IF (seq.Step(inStepID := seq.RESTORE_STEP_ID,
    inEnabled := TRUE,
    inStepDescription := 'RETURN TO THE START OF THE SEQUENCE')) THEN
    //--------------------------------------------------------	
		refSequenceTask.DoneWhen(TRUE);
    	seq.CompleteSequence();
    //--------------------------------------------------------			
END_IF;


IF refSequenceTask.HandleTaskError() THEN
	//here we can decide what to do
	//	refSequenceTask.Restore();
	_feedNewBlisterTask.Restore();
END_IF



seq.Close();
END_METHOD

METHOD PRIVATE SequenceOutgoingBlister
VAR_INPUT
	refSequenceTask : REFERENCE TO TcoFeedingSequenceTask;
	
	
END_VAR

VAR
    seq    : REFERENCE TO TcoCore.TcoSequence;

END_VAR

VAR_INST
	_timer:ton;
	
END_VAR
seq REF= refSequenceTask.Sequence;
refSequenceTask(inoStatus:=_status,inoConfig:=_config);

seq.Open();
seq.Observer := refSequenceTask.Observer;



		



//***************************************************************************************************     
//    This step will be executed and immediately finished, as the condition in Await method is true.
IF seq.Step(0,TRUE,'<#INIT#>') THEN   
	Messenger.Warning('<#BEZPECNOST ZARIADENIA NARUSENA. NIEJE MOZNE VYKONAT AKCIU#>');     
	IF _status.SafeCondition THEN
    	seq.CompleteStep();
	END_IF;
END_IF        
//***************************************************************************************************     

IF seq.Step(10,TRUE,'<#SEPAROVANIE VYSTUPNEHO BLISTRA - UVOLNENIE BLISTRA VYSUNUTIE P9#>') THEN   

    seq.StepCompleteWhen( (THIS^.Components.P9_LockEntryBlisterTop.MoveToWork().Done OR _config.LockBlisterInPickPosInactive) AND THIS^.Components.P8_FixEntryBlisterSide.MoveToHome().Done);
END_IF        
//***************************************************************************************************   


//***************************************************************************************************     
IF seq.Step(20,TRUE,'<#SEPAROVANIE VYSTUPNEHO BLISTRA - ZASUNUTIE SUPPORTU P7#>') THEN   

   seq.StepCompleteWhen(THIS^.Components.P7_SupportEntryBlister.MoveToHome().Done);
END_IF        
//***************************************************************************************************   



//***************************************************************************************************     
IF seq.Step(30,TRUE,'<#SEPAROVANIE VYSTUPNEHO BLISTRA - KONTROLA PRITOMNOSTI BLISTA NA SKLZE (I5) #>') THEN   
	IF seq.IsFreshState THEN
		_timer(IN:=FALSE);
	END_IF
	_timer(IN:=THIS^.Components.I5_OutBlistersIsThrowedCorrectly.Signal,PT:=_config.StabilisationTime);
	
    seq.StepCompleteWhen(_timer.Q);
	
	IF Components.P4_FeedEntryBlister.AtHome AND NOT THIS^.Components.I5_OutBlistersIsThrowedCorrectly.Signal THEN
		seq.StepCompleteWhen(seq.CurrentStep.Duration>_config.StabilisationTime);
	END_IF
END_IF        
//***************************************************************************************************   



IF (seq.Step(inStepID := seq.RESTORE_STEP_ID,
    inEnabled := TRUE,
    inStepDescription := 'RETURN TO THE START OF THE SEQUENCE')) THEN
    //--------------------------------------------------------	
		refSequenceTask.DoneWhen(TRUE);
    	seq.CompleteSequence();
    //--------------------------------------------------------			
END_IF;


IF refSequenceTask.HandleTaskError() THEN
	//here we can decide what to do
	//	refSequenceTask.Restore();
	_throwBlisterTask.Restore();


END_IF


seq.Close();
END_METHOD

METHOD PRIVATE SequenceOutgoingBuffer
VAR_INPUT
	refSequenceTask : REFERENCE TO TcoFeedingSequenceTask;
	
	
END_VAR

VAR
    seq    : REFERENCE TO TcoCore.TcoSequence;

END_VAR

VAR_INST
	_timer:ton;
	
END_VAR
seq REF= refSequenceTask.Sequence;
refSequenceTask(inoStatus:=_status,inoConfig:=_config);

seq.Open();
seq.Observer := refSequenceTask.Observer;



		



//***************************************************************************************************     
//    This step will be executed and immediately finished, as the condition in Await method is true.
IF seq.Step(0,TRUE,'<#INIT#>') THEN   
	Messenger.Warning('<#BEZPECNOST ZARIADENIA NARUSENA. NIEJE MOZNE VYKONAT AKCIU#>');     
	IF _status.SafeCondition THEN
    	seq.CompleteStep();
	END_IF;
END_IF        
//***************************************************************************************************     



//***************************************************************************************************     
IF seq.Step(10,TRUE,'<#VYSTUPNY BUFFER - KONTROLA PRITOMNOSTI BLISTA NAD BUFFEROM  #>') THEN   
	IF seq.IsFreshState THEN
		_timer(IN:=FALSE);
	END_IF
	_timer(IN:=(*NOT THIS^.Components.I5_OutBlistersIsThrowedCorrectly.Signal AND*) Components.I7_OutBlistersIsAboveOutBuffer.Signal,PT:=_config.StabilisationTime);
	
    seq.StepCompleteWhen(_timer.Q);
END_IF        
//***************************************************************************************************   


//***************************************************************************************************     
IF seq.Step(20,TRUE,'<#VYSTUPNY BUFFER - KONTROLA POSCTU BLISTROV SNIMAC I8 #>') THEN   
	Messenger.Warning('<#PODAVAC PLNY! ODSTRANTE PRAZDNE BLISTRE (I8) !#>');
    seq.StepCompleteWhen(THIS^.Components.I8_OutBlistersBufferIsFull.IsFalse);
END_IF        
//***************************************************************************************************   


//***************************************************************************************************     
IF seq.Step(30,TRUE,'<#VYSTUPNY BUFFER - P6 POSUN KUSOV NAD BUFFER#>') THEN   

	THIS^.Components.P6_VerticalSepareOutBlister.MoveToWork();
	IF Components.I6_OutBlistersLisftSignal.Signal THEN
	
		THIS^.Components.P6_VerticalSepareOutBlister.MoveWorkTask.Abort();
	    seq.StepCompleteWhen(TRUE);
	END_IF;
		
END_IF        
//***************************************************************************************************   


//***************************************************************************************************     
IF seq.Step(40,TRUE,'<#VYSTUPNY BUFFER - UVOLNENIE BLISTRA  P5 PRACOVNA POZICIA #>') THEN   

	
	seq.StepCompleteWhen(Components.P5_HorizontalSepareOutBlisters.MoveToWork().Done);
		
END_IF        
//***************************************************************************************************   

//***************************************************************************************************     
IF seq.Step(45,TRUE,'<#VYSTUPNY BUFFER - P6 NAVRAT NAHOR#>') THEN   

	
	seq.StepCompleteWhen( THIS^.Components.P6_VerticalSepareOutBlister.MoveToHome().Done);
		
END_IF        
//***************************************************************************************************   

//***************************************************************************************************     
IF seq.Step(50,TRUE,'<#VYSTUPNY BUFFER - HORIZONTALNE ZASUNUTIE P5 ZAKLADNA POZICIA#>') THEN   

	
	seq.StepCompleteWhen(Components.P5_HorizontalSepareOutBlisters.MoveToHome().Done);
		
END_IF        
//***************************************************************************************************   



IF (seq.Step(inStepID := seq.RESTORE_STEP_ID,
    inEnabled := TRUE,
    inStepDescription := 'RETURN TO THE START OF THE SEQUENCE')) THEN
    //--------------------------------------------------------	
		refSequenceTask.DoneWhen(TRUE);
    	seq.CompleteSequence();
    //--------------------------------------------------------			
END_IF;


IF refSequenceTask.HandleTaskError() THEN
	//here we can decide what to do
	//refSequenceTask.Restore();
	_hanldeOutBufferTask.Restore();
END_IF


seq.Close();
END_METHOD

METHOD PRIVATE SequenceResetToDefault
VAR_INPUT
	refSequenceTask : REFERENCE TO TcoFeedingSequenceTask;
	
	
END_VAR

VAR
    seq    : REFERENCE TO TcoCore.TcoSequence;

END_VAR

VAR_INST
	_timer:ton;
	
END_VAR
seq REF= refSequenceTask.Sequence;
refSequenceTask(inoStatus:=_status,inoConfig:=_config);
seq.Open();
seq.Observer := refSequenceTask.Observer;



		



//***************************************************************************************************     
//    This step will be executed and immediately finished, as the condition in Await method is true.
IF seq.Step(0,TRUE,'<#INIT#>') THEN   
	Messenger.Warning('<#BEZPECNOST ZARIADENIA NARUSENA. NIEJE MOZNE VYKONAT AKCIU#>');     
	IF _status.SafeCondition THEN
    	seq.CompleteStep();
	END_IF;
END_IF        
//***************************************************************************************************     



//***************************************************************************************************     
IF seq.Step(10,TRUE,'<#VYCHODIZA POLOHA - VYSUNUTIE P3#>') THEN   

    seq.StepCompleteWhen(Components.P3_HorizontalSepareEntryBlisters.MoveToWork().Done );
END_IF        
//***************************************************************************************************   


//***************************************************************************************************     
IF seq.Step(20,NOT _config.SepareBlistersAtEntryInactive,'<#VYCHODIZA POLOHA - ZASUNUTIE P10#>') THEN   

    seq.StepCompleteWhen(Components.P10_HoldEntrySepareOutBlister.MoveToHome().Done);
END_IF        
//***************************************************************************************************   


//***************************************************************************************************     
IF seq.Step(30,TRUE,'<#VYCHODIZA POLOHA - ZASUNUTIE P1 A P2>') THEN   


	    seq.StepCompleteWhen(Components.P1_VerticalSepareEntryBlisters.MoveToHome().Done AND_THEN Components.P2_VerticalSepareEntryBlisters.MoveToHome().Done);

END_IF        
//***************************************************************************************************   


//***************************************************************************************************     
IF seq.Step(40,TRUE,'<#VYCHODIZA POLOHA - ZASUNUTIE P5#>') THEN   

	
	seq.StepCompleteWhen(Components.P5_HorizontalSepareOutBlisters.MoveToHome().Done);
		
END_IF        
//***************************************************************************************************   

//***************************************************************************************************     
IF seq.Step(50,TRUE,'<#VYCHODIZA POLOHA - ZASUNUTIE P6#>') THEN   

	
	seq.StepCompleteWhen(Components.P6_VerticalSepareOutBlister.MoveToHome().Done);
		
END_IF        
//***************************************************************************************************   

//***************************************************************************************************     
IF seq.Step(60,TRUE,'<#VYCHODIZA POLOHA - ZASUNUTIE P4 DO ZAKLADNEJ POZICIE#>') THEN   

	
	seq.StepCompleteWhen(Components.P4_FeedEntryBlister.MoveToHome().Done);
		
END_IF        
//***************************************************************************************************   

//***************************************************************************************************     
IF seq.Step(70,COmponents.I4_PresentBlisterInWorkingPos.Signal AND
				Components.P8_FixEntryBlisterSide.AtWork,'<#SEPAROVANIE VSTUPNEHO BLISTRA - PODoPRETIE  A ZAFIXOVANIE KUSU P7 VYSUNT A P9 ZASUNUT #>') THEN   

    seq.StepCompleteWhen(THIS^.Components.P7_SupportEntryBlister.MoveToWork().Done AND (THIS^.Components.P9_LockEntryBlisterTop.MoveToHome().Done OR _config.LockBlisterInPickPosInactive));
END_IF        
//***************************************************************************************************   


IF (seq.Step(inStepID := seq.RESTORE_STEP_ID,
    inEnabled := TRUE,
    inStepDescription := 'RETURN TO THE START OF THE SEQUENCE')) THEN
    //--------------------------------------------------------	
		refSequenceTask.DoneWhen(TRUE);
    	seq.CompleteSequence();
    //--------------------------------------------------------			
END_IF;



IF refSequenceTask.HandleTaskError() THEN
	
	//here we can decide what to do
	//	refSequenceTask.Restore();

END_IF

seq.Close();
END_METHOD

(*~
	<docu>
		<summary>
		    Custom service (manual, maintenance) logic.
			This method must be implemented in derived class.
		</summary>			
	</docu>	
~*)
METHOD PROTECTED  ServiceMode
_components.Q3_AttentionSignalisationB.Service();
_components.Q2_AttentionSignalisationG.Service();
_components.Q1_AttentionSignalisationR.Service();
_components.P1_VerticalSepareEntryBlisters.Service();
_components.P2_VerticalSepareEntryBlisters.Service();
_components.P3_HorizontalSepareEntryBlisters.Service();
_components.P4_FeedEntryBlister.Service();
_components.P5_HorizontalSepareOutBlisters.Service();
_components.P6_VerticalSepareOutBlister.Service();
_components.P7_SupportEntryBlister.Service();
_components.P8_FixEntryBlisterSide.Service();
_components.P9_LockEntryBlisterTop.Service();
_components.P10_HoldEntrySepareOutBlister.Service();
END_METHOD

PROPERTY PUBLIC SetSequencesToStep : bool
GET
SetSequencesToStep:=_setSequencesToStep;
END_GET
SET
_setSequencesToStep:=SetSequencesToStep;
END_SET
END_PROPERTY

METHOD PUBLIC SetToDefault : TcoCore.ITcoTaskStatus
SetToDefault := _setToDefaultTask.Invoke();
END_METHOD

PROPERTY SetToDefaultTask : REFERENCE TO TcoFeedingSequenceTask
GET
SetToDefaultTask ref=_setToDefaultTask;
END_GET
END_PROPERTY

(*~
	<docu>
		<summary>
			Gets the status of the MTS Pls feeder. 					
		</summary>			
	</docu>	
~*)
PROPERTY Status : REFERENCE TO TcoPlsPaletizator_Status_v_1_x_x
GET
Status REF= _status;
END_GET
END_PROPERTY

METHOD PUBLIC ThrowBlister : TcoCore.ITcoTaskStatus

ThrowBlister := _throwBlisterTask.Invoke();
END_METHOD

PROPERTY ThrowBlisterTask : REFERENCE TO TcoFeedingSequenceTask
GET
ThrowBlisterTask ref=_throwBlisterTask;
END_GET
END_PROPERTY

END_FUNCTION_BLOCK

// ---- Abstractions/Components/MtsFeeding/Components/OscilatingConveyorFeeder/TcoOscilatingConveyorFeeder.TcPOU
FUNCTION_BLOCK TcoOscilatingConveyorFeeder EXTENDS TcoCore.TcoComponent
VAR_INPUT
    inSafeCondition : BOOL;
    inDoorOpen : BOOL;
    inMOde : eCUMode;
END_VAR

VAR_OUTPUT
END_VAR
VAR
    {attribute addProperty Name "<#Config#>"}
    _config : TcoOscilatingConveyorFeeder_Config_v_1_x_x;
    {attribute addProperty Name "<#Status#>"}
    {attribute clr [ReadOnly()]}
    _status : TcoOscilatingConveyorFeeder_Status_v_1_x_x;
    {attribute addProperty Name "<#Control#>"}
    _control : TcoOscilatingConveyorFeeder_Control_v_1_x_x;

    {attribute addProperty Name "<#Components#>"}
    _components : TcoOscilatingConveyorFeederComponents := (Parent := THIS^);

    {attribute addProperty Name "<#Poziadavka separovania#>"}
    _feedComponentsTask : TcoFeedingSequenceTask(THIS^);
    {attribute addProperty Name "<#Poziadavka vyprazdnenia#>"}
    _throwCompoentsTask : TcoFeedingSequenceTask(THIS^);

    {attribute addProperty Name "<#Poziadavka vychodzej polohy#>"}
    _setToDefaultTask : TcoFeedingSequenceTask(THIS^);

    {attribute addProperty Name "<#Restore#>"}
    _restoreTask : TcoCore.TcoTask(THIS^);

    {attribute clr [CompilerOmits("BuilderPlainer", "BuilderOnliner","BuilderOnlinerInterface","BuilderShadowerInterface")]}
    _blinker : TcoBlinker(THIS^);
    _timerEntryEmpty : ton;
    _timerOutFull : ton;
    _timerDisableSafety : TON;
    {attribute addProperty Name "<#Temporarily disabled safety#>"}
    _temporarilyDisableSafety : BOOL;

    {attribute clr [CompilerOmits("BuilderPlainer", "BuilderOnliner","BuilderOnlinerInterface","BuilderShadowerInterface")]}
    restoreDone : BOOL;
    {attribute clr [CompilerOmits("BuilderPlainer", "BuilderOnliner","BuilderOnlinerInterface","BuilderShadowerInterface")]}
    _setSequencesToStep : BOOL := FALSE;

    {attribute addProperty Name "<#Oscilating Specific Data#>"}
    _specificData : TcoOscilatingConveyorFeeder_DesignerSpecificData(THIS^);
END_VAR

_status.SafeCondition := inSafeCondition;
_status.EntryBufferEmpty := not Components.iEntryFeederIsEmpty.Signal;

_components.Designer(inoData := _specificData);

_status.PcToPlcData := _specificData.PcToPlcData;

IF _config.ControledByVisonSystem THEN
    //send states to vision system
    _specificData.PlcToPcData.Config := _config;
    _specificData.PlcToPcData.SafeCondition := inSafeCondition;
    _specificData.PlcToPcData.DoorOpen := inDoorOpen;
    _specificData.PlcToPcData.Mode := inMOde;
    _specificData.PlcToPcData.EntryFeederError := _components.iEntryFeederError.Signal;
    _specificData.PlcToPcData.EntryFeederIsEmpty := _components.iEntryFeederIsEmpty.Signal;
    _specificData.PlcToPcData.FlowSensor := _components.iFlowSensor.Signal;
    _specificData.PlcToPcData.OscConvError := _components.iOscConvError.Signal;
    _specificData.PlcToPcData.ThrowBoxPresent := _components.iThrowBoxPresent.Signal;
    _specificData.PlcToPcData.SideGuardAtHome := _components.SideGuard.AtHome;
    _specificData.PlcToPcData.SideGuardAtWork := _components.SideGuard.AtWork;

    //listen vision system
    _components.qOscConvRun.Reset();
    IF _specificData.PcToPlcData.OscConvRun THEN
        _components.qOscConvRun.Set();
    END_IF;

    _components.qOscConvRunReverse.Reset();
    IF _specificData.PcToPlcData.OscConvRunReverse THEN
        _components.qOscConvRunReverse.Set();
    END_IF;

    _components.qEntryFeederRun.Reset();
    IF _specificData.PcToPlcData.EntryFeederRun THEN
        _components.qEntryFeederRun.Set();
    END_IF;

    _components.qOscCylinderRow1Left.Reset();
    IF _specificData.PcToPlcData.OscCylinderRow1Left THEN
        _components.qOscCylinderRow1Left.Set();
    END_IF;

    _components.qOscCylinderRow1Middle.Reset();
    IF _specificData.PcToPlcData.OscCylinderRow1Middle THEN
        _components.qOscCylinderRow1Middle.Set();
    END_IF;

    _components.qOscCylinderRow1Right.Reset();
    IF _specificData.PcToPlcData.OscCylinderRow1Right THEN
        _components.qOscCylinderRow1Right.Set();
    END_IF;

    _components.qOscCylinderRow2Left.Reset();
    IF _specificData.PcToPlcData.OscCylinderRow2Left THEN
        _components.qOscCylinderRow2Left.Set();
    END_IF;

    _components.qOscCylinderRow2Middle.Reset();
    IF _specificData.PcToPlcData.OscCylinderRow2Middle THEN
        _components.qOscCylinderRow2Middle.Set();
    END_IF;

    _components.qOscCylinderRow2Right.Reset();
    IF _specificData.PcToPlcData.OscCylinderRow2Right THEN
        _components.qOscCylinderRow2Right.Set();
    END_IF;

    _components.qOscCylinderRow3Left.Reset();
    IF _specificData.PcToPlcData.OscCylinderRow3Left THEN
        _components.qOscCylinderRow3Left.Set();
    END_IF;

    _components.qOscCylinderRow3Middle.Reset();
    IF _specificData.PcToPlcData.OscCylinderRow3Middle THEN
        _components.qOscCylinderRow3Middle.Set();
    END_IF;

    _components.qOscCylinderRow3Right.Reset();
    IF _specificData.PcToPlcData.OscCylinderRow3Right THEN
        _components.qOscCylinderRow3Right.Set();
    END_IF;

    IF _config.EnableSideGuard THEN
        IF _specificData.PcToPlcData.SideGuard THEN
            _components.SideGuard.MoveHomeTask.Restore();
            _components.SideGuard.MoveToWork();
        ELSE
            _components.SideGuard.MoveWorkTask.Restore();
            _components.SideGuard.MoveToHome();
        END_IF
    END_IF;

    IF _config.EnableEntryFeederMantinel THEN
        IF _specificData.PcToPlcData.EntryFeederMantinel THEN
            _components.EntryFeederMantinel.MoveHomeTask.Restore();
            _components.EntryFeederMantinel.MoveToWork();
        ELSE
            _components.EntryFeederMantinel.MoveWorkTask.Restore();
            _components.EntryFeederMantinel.MoveToHome();
        END_IF
    END_IF;

ELSE

    IF _config.StepModeManagableFromOutside THEN
        IF _setSequencesToStep THEN
            _feedComponentsTask.SetStepMode();
            _throwCompoentsTask.SetStepMode();
            _setToDefaultTask.SetStepMode();
        ELSE
            _feedComponentsTask.SetCyclicMode();
            _throwCompoentsTask.SetCyclicMode();
            _setToDefaultTask.SetCyclicMode();
        END_IF
    END_IF;

    _feedComponentsTask.Enabled := NOT _throwCompoentsTask.Busy;
    IF (_feedComponentsTask.Execute()) THEN
        SequenceIncomingBlister(refSequenceTask := _feedComponentsTask);
    END_IF;

    _throwCompoentsTask.Enabled := NOT _feedComponentsTask.Busy;
    IF (_throwCompoentsTask.Execute()) THEN
        SequenceOutgoingBlister(refSequenceTask := _throwCompoentsTask);
    END_IF;

    _setToDefaultTask.Enabled := TRUE;
    IF (_setToDefaultTask.Execute()) THEN
        SequenceResetToDefault(refSequenceTask := _setToDefaultTask);
    END_IF;

END_IF

//*************RESTORE********************

_restoreTask.Enabled := TRUE;

IF _restoreTask.Execute() THEN
    Restore();
    _restoreTask.DoneWhen(inCondition := TRUE);
END_IF

//****************************************

//********************SAFETY******************
_timerDisableSafety(IN := _temporarilyDisableSafety, PT := _config.TimeToDisableSafety);

THIS^.Messenger.OnCondition(inCondition := _temporarilyDisableSafety).Warning('SAFTY TEMPORARILY DISABLED!');

IF NOT _temporarilyDisableSafety THEN
    IF NOT _status.SafeCondition THEN
        _components.qOscConvRun.Reset();
        _components.qOscConvRunReverse.Reset();
        _components.qOscCylinderRow1Left.Reset();
        _components.qOscCylinderRow1Middle.Reset();
        _components.qOscCylinderRow1Right.Reset();

        _components.qOscCylinderRow2Left.Reset();
        _components.qOscCylinderRow2Middle.Reset();
        _components.qOscCylinderRow2Right.Reset();

        _components.qOscCylinderRow3Left.Reset();
        _components.qOscCylinderRow3Middle.Reset();
        _components.qOscCylinderRow3Right.Reset();

    END_IF

END_IF;

IF _timerDisableSafety.Q THEN
    _temporarilyDisableSafety := FALSE;
END_IF

PROPERTY Components : REFERENCE TO TcoOscilatingConveyorFeederComponents
GET
Components ref=_components;
END_GET
END_PROPERTY

(*~
	<docu>
		<summary>
			Gets the configuration of the MTS Oscilating conveyor feeder. 					
		</summary>			
	</docu>	
~*)
PROPERTY Config : REFERENCE TO TcoOscilatingConveyorFeeder_Config_v_1_x_x
GET
Config REF= _config;
END_GET
END_PROPERTY

METHOD PUBLIC DefaultSignalisation
VAR_INPUT
END_VAR
Components.Q1_AttentionSignalisationR.Reset();
Components.Q2_AttentionSignalisationG.Reset();
Components.Q3_AttentionSignalisationB.Reset();

_blinker(inOffTime:=_config.BlinkTime,inOnTime:=_config.BlinkTime);
_timerEntryEmpty(in:= _status.EntryBufferEmpty,Pt:=_config.InfoTime);
//_timerOutFull(in:=  _status.OutBufferFull ,Pt:=_config.InfoTime);
IF NOT inDoorOpen  
	AND NOT _timerEntryEmpty.Q
	AND NOT _timerOutFull.q THEN
	Components.Q2_AttentionSignalisationG.Set();
ELSIF  _blinker.IsOn THEN
	IF inDoorOpen AND 
		(
		THIS^._feedComponentsTask.Busy
		OR
		THIS^._throwCompoentsTask.Busy
		 )THEN
		Messenger.Warning('<#CAKANIE NA OBSLUHU PALETIZERA - ZAVRITE DVERE!#>');
		Components.Q1_AttentionSignalisationR.Set();
		Components.Q2_AttentionSignalisationG.Set();
	ELSIF _timerEntryEmpty.Q
		THEN
		Components.Q1_AttentionSignalisationR.Set();
		Components.Q2_AttentionSignalisationG.Set();
	ELSIF _timerOutFull.Q
		THEN
		
		Components.Q1_AttentionSignalisationR.Set();
		Components.Q2_AttentionSignalisationG.Set();

//	ELSIF NOT _status.OutBufferFull
//		AND _status.EntryBufferEmpty 
//		AND NOT _status.BlisterReady THEN	
//		Components.Q1_AttentionSignalisationR.Set();
//	ELSIF  _status.OutBufferFull  THEN
//		Components.Q1_AttentionSignalisationR.Set();	
	
	END_IF;


	
END_IF;
END_METHOD

PROPERTY FeedComponentsTask : REFERENCE TO TcoFeedingSequenceTask
GET
FeedComponentsTask ref=_feedComponentsTask;
END_GET
END_PROPERTY

METHOD PUBLIC FeedNewComponents : TcoCore.ITcoTaskStatus
FeedNewComponents := _feedComponentsTask.Invoke();
END_METHOD

(*~
	<docu>
		<summary>
			Restores this instance to the Ready state. Can be called explicitly or from within one of the restore mechanisms.	
		</summary>			
	</docu>	
~*)
METHOD  Restore : ITcoRestorable

_feedComponentsTask.Restore();
_throwCompoentsTask.Restore();
_setToDefaultTask.Restore();
_messenger.UnPin();
END_METHOD

METHOD PRIVATE SequenceIncomingBlister
VAR_INPUT
	refSequenceTask : REFERENCE TO TcoFeedingSequenceTask;
	
	
END_VAR

VAR
    seq    : REFERENCE TO TcoCore.TcoSequence;


END_VAR
seq REF= refSequenceTask.Sequence;
refSequenceTask(inoStatus:=_status,inoConfig:=_config);


seq.Open();
seq.Observer := refSequenceTask.Observer;



		



//***************************************************************************************************     
//    This step will be executed and immediately finished, as the condition in Await method is true.
IF seq.Step(0,TRUE,'<#INIT#>') THEN   
	Messenger.Warning('<#BEZPECNOST ZARIADENIA NARUSENA. NIEJE MOZNE VYKONAT AKCIU#>');     
	IF _status.SafeCondition THEN
    	seq.CompleteStep();
	END_IF;
END_IF        
//***************************************************************************************************     

 
////***************************************************************************************************     
//IF seq.Step(10,TRUE,'<#KONTROLA POCTU VSTUPNYCH BLISTROV#>') THEN   
//    Messenger.Warning('<#PODAVAC PRAZDNY! DOPLNE VSTUPNE BLISTRE !#>');
//    seq.StepCompleteWhen(Components.I3_PresentBlistersInBufferEmpty.IsTrue);
//END_IF        
////***************************************************************************************************     


        
////***************************************************************************************************     
//IF seq.Step(20,TRUE,'<#SEPAROVANIE VSTUPNEHO BLISTRA - VERTIKALNE VALCE VYSUNUTE P1 A P2 #>') THEN   

//    seq.StepCompleteWhen(THIS^.Components.P1_VerticalSepareEntryBlisters.MoveToWork().Done AND THIS^.Components.P2_VerticalSepareEntryBlisters.MoveToWork().Done);
//END_IF        
////***************************************************************************************************     


////***************************************************************************************************     
//IF seq.Step(30,TRUE,'<#SEPAROVANIE VSTUPNEHO BLISTRA - SEPAROVANIE ZASUNUTE P3#>') THEN   

//    seq.StepCompleteWhen(THIS^.Components.P3_HorizontalSepareEntryBlisters.MoveToHome().Done);
//END_IF        
////***************************************************************************************************     


////***************************************************************************************************     
//IF seq.Step(40,TRUE,'<#SEPAROVANIE VSTUPNEHO BLISTRA - VERTIKALNE VALCE  ZASUNUT P1#>') THEN   

//    seq.StepCompleteWhen(THIS^.Components.P1_VerticalSepareEntryBlisters.MoveToHome().Done );
//END_IF        
////***************************************************************************************************     

////***************************************************************************************************     
//IF seq.Step(45,TRUE,'<#SEPAROVANIE VSTUPNEHO BLISTRA - VERTIKALNE VALCE VYSUNUT P2#>') THEN   

//    seq.StepCompleteWhen( THIS^.Components.P2_VerticalSepareEntryBlisters.MoveToWork().Done);
//END_IF        
////***************************************************************************************************     


////***************************************************************************************************     
//IF seq.Step(50,TRUE,'<#SEPAROVANIE VSTUPNEHO BLISTRA - SEPAROVANIE VYSUNUTE P3 A P10#>') THEN   

//    seq.StepCompleteWhen(THIS^.Components.P3_HorizontalSepareEntryBlisters.MoveToWork().Done AND (Components.P10_HoldEntrySepareOutBlister.MoveToWork().Done or _config.SepareBlistersAtEntryInactive));
//END_IF        
////***************************************************************************************************     

////***************************************************************************************************     
//IF seq.Step(60,TRUE,'<#SEPAROVANIE VSTUPNEHO BLISTRA - VERTIKALNE VALCE ZASUNUT P1 A P@#>') THEN   

//    seq.StepCompleteWhen(THIS^.Components.P1_VerticalSepareEntryBlisters.MoveToHome().Done AND THIS^.Components.P2_VerticalSepareEntryBlisters.MoveToHome().Done); 
					
//END_IF        
////***************************************************************************************************     

////***************************************************************************************************     
//IF seq.Step(65,NOT _config.SepareBlistersAtEntryInactive,'<#SEPAROVANIE VSTUPNEHO BLISTRA - ZASUNUTIE P10>') THEN   

//    seq.StepCompleteWhen(Components.P10_HoldEntrySepareOutBlister.MoveToHome().Done  );
//END_IF        
////***************************************************************************************************     

////***************************************************************************************************   
//IF seq.Step(70,TRUE,'<#KONTROLA PRITOMNOSTI SEPAROVANEHO KUSU#>') THEN   
//    Messenger.Error('<#PODAVAC PRAZDNY! DOPLNE BLISTRE !#>');
//    seq.StepCompleteWhen(THIS^.Components.I1_PresentBlisterEntry.IsTrue AND (THIS^.Components.I2_PresentBlisterEntryEmptySpace.IsTrue) );
//END_IF        
////***************************************************************************************************     


////***************************************************************************************************     
//IF seq.Step(80,TRUE,'<#SEPAROVANIE VSTUPNEHO BLISTRA - UPEVNENIE BLISTRA ZASUNUT P8#>') THEN   

//    seq.StepCompleteWhen(THIS^.Components.P8_FixEntryBlisterSide.MoveToHome().Done);
//END_IF        
////***************************************************************************************************     

////***************************************************************************************************     
//IF seq.Step(85,TRUE,'<#SEPAROVANIE VSTUPNEHO BLISTRA - CAKANIE NA PRESUNUTIE BLISTRA DO ODOBERACEJ POLOHY P4 A I1 #>') THEN   

//    seq.StepCompleteWhen(THIS^.Components.P4_FeedEntryBlister.MoveToWork().Done AND Components.i4_PresentBlisterInWorkingPos.IsTrue);
//END_IF        
////***************************************************************************************************     


////***************************************************************************************************     
//IF seq.Step(90,TRUE,'<#SEPAROVANIE VSTUPNEHO BLISTRA - UPEVENIE BLISTRA ZBOKU#>') THEN   

//    seq.StepCompleteWhen(THIS^.Components.P8_FixEntryBlisterSide.MoveToWork().Done);
//END_IF        
////***************************************************************************************************     



////***************************************************************************************************     
//IF seq.Step(100,TRUE,'<#SEPAROVANIE VSTUPNEHO BLISTRA - NPRESUNUTIE BLISTRA DO POZICIE NABERANIA#>') THEN   

//   IF THIS^.Components.P6_VerticalSepareOutBlister.AtHome THEN
//	    seq.CompleteStep();
//	ELSE
//		Messenger.Error('VYSTUPNY BUFFER NIEJE V HORNEJ POZICII!(P6)');
//	END_IF
//END_IF        
////***************************************************************************************************   

////***************************************************************************************************     
//IF seq.Step(110,TRUE,'<#SEPAROVANIE VSTUPNEHO BLISTRA - ZASUNUTE P4#>') THEN   

//	 seq.StepCompleteWhen(THIS^.Components.P4_FeedEntryBlister.MoveToHome().Done) ;
	
//END_IF        
////***************************************************************************************************   


////***************************************************************************************************     
//IF seq.Step(120,TRUE,'<#SEPAROVANIE VSTUPNEHO BLISTRA - PODoPRETIE  A ZAFIXOVANIE KUSU P7 VYSUNT A P9 ZASUNUT #>') THEN   

//    seq.StepCompleteWhen(THIS^.Components.P7_SupportEntryBlister.MoveToWork().Done AND (THIS^.Components.P9_LockEntryBlisterTop.MoveToHome().Done OR _config.LockBlisterInPickPosInactive));
//END_IF        
////***************************************************************************************************   




IF (seq.Step(inStepID := seq.RESTORE_STEP_ID,
    inEnabled := TRUE,
    inStepDescription := 'RETURN TO THE START OF THE SEQUENCE')) THEN
    //--------------------------------------------------------	
		refSequenceTask.DoneWhen(TRUE);
    	seq.CompleteSequence();
    //--------------------------------------------------------			
END_IF;


IF refSequenceTask.HandleTaskError() THEN
	//here we can decide what to do
	//	refSequenceTask.Restore();
	_feedComponentsTask.Restore();
END_IF



seq.Close();
END_METHOD

METHOD PRIVATE SequenceOutgoingBlister
VAR_INPUT
	refSequenceTask : REFERENCE TO TcoFeedingSequenceTask;
	
	
END_VAR

VAR
    seq    : REFERENCE TO TcoCore.TcoSequence;

END_VAR

VAR_INST
	_timer:ton;
	
END_VAR
seq REF= refSequenceTask.Sequence;
refSequenceTask(inoStatus:=_status,inoConfig:=_config);

seq.Open();
seq.Observer := refSequenceTask.Observer;



		



//***************************************************************************************************     
//    This step will be executed and immediately finished, as the condition in Await method is true.
IF seq.Step(0,TRUE,'<#INIT#>') THEN   
	Messenger.Warning('<#BEZPECNOST ZARIADENIA NARUSENA. NIEJE MOZNE VYKONAT AKCIU#>');     
	IF _status.SafeCondition THEN
    	seq.CompleteStep();
	END_IF;
END_IF        
//***************************************************************************************************     

//IF seq.Step(10,TRUE,'<#SEPAROVANIE VYSTUPNEHO BLISTRA - UVOLNENIE BLISTRA VYSUNUTIE P9#>') THEN   

//    seq.StepCompleteWhen( (THIS^.Components.P9_LockEntryBlisterTop.MoveToWork().Done OR _config.LockBlisterInPickPosInactive) AND THIS^.Components.P8_FixEntryBlisterSide.MoveToHome().Done);
//END_IF        
////***************************************************************************************************   


////***************************************************************************************************     
//IF seq.Step(20,TRUE,'<#SEPAROVANIE VYSTUPNEHO BLISTRA - ZASUNUTIE SUPPORTU P7#>') THEN   

//   seq.StepCompleteWhen(THIS^.Components.P7_SupportEntryBlister.MoveToHome().Done);
//END_IF        
////***************************************************************************************************   



////***************************************************************************************************     
//IF seq.Step(30,TRUE,'<#SEPAROVANIE VYSTUPNEHO BLISTRA - KONTROLA PRITOMNOSTI BLISTA NA SKLZE (I5) #>') THEN   
//	IF seq.IsFreshState THEN
//		_timer(IN:=FALSE);
//	END_IF
//	_timer(IN:=THIS^.Components.I5_OutBlistersIsThrowedCorrectly.Signal,PT:=_config.StabilisationTime);
	
//    seq.StepCompleteWhen(_timer.Q);
	
//	IF Components.P4_FeedEntryBlister.AtHome AND NOT THIS^.Components.I5_OutBlistersIsThrowedCorrectly.Signal THEN
//		seq.StepCompleteWhen(seq.CurrentStep.Duration>_config.StabilisationTime);
//	END_IF
//END_IF        
////***************************************************************************************************   



IF (seq.Step(inStepID := seq.RESTORE_STEP_ID,
    inEnabled := TRUE,
    inStepDescription := 'RETURN TO THE START OF THE SEQUENCE')) THEN
    //--------------------------------------------------------	
		refSequenceTask.DoneWhen(TRUE);
    	seq.CompleteSequence();
    //--------------------------------------------------------			
END_IF;


IF refSequenceTask.HandleTaskError() THEN
	//here we can decide what to do
	//	refSequenceTask.Restore();
	_throwCompoentsTask.Restore();


END_IF


seq.Close();
END_METHOD

METHOD PRIVATE SequenceResetToDefault
VAR_INPUT
	refSequenceTask : REFERENCE TO TcoFeedingSequenceTask;
	
	
END_VAR

VAR
    seq    : REFERENCE TO TcoCore.TcoSequence;

END_VAR

VAR_INST
	_timer:ton;
	
END_VAR
seq REF= refSequenceTask.Sequence;
refSequenceTask(inoStatus:=_status,inoConfig:=_config);
seq.Open();
seq.Observer := refSequenceTask.Observer;



		



//***************************************************************************************************     
//    This step will be executed and immediately finished, as the condition in Await method is true.
IF seq.Step(0,TRUE,'<#INIT#>') THEN   
	Messenger.Warning('<#BEZPECNOST ZARIADENIA NARUSENA. NIEJE MOZNE VYKONAT AKCIU#>');     
	IF _status.SafeCondition THEN
    	seq.CompleteStep();
	END_IF;
END_IF        
//***************************************************************************************************     



//***************************************************************************************************     
IF seq.Step(10,TRUE,'<#VYCHODIZA POLOHA - VYPNUTIE VALCOV#>') THEN   
		_components.qOscCylinderRow1Left.Reset();
		_components.qOscCylinderRow1Middle.Reset();
		_components.qOscCylinderRow1Right.Reset();

		_components.qOscCylinderRow2Left.Reset();
		_components.qOscCylinderRow2Middle.Reset();
		_components.qOscCylinderRow2Right.Reset();

		_components.qOscCylinderRow3Left.Reset();
		_components.qOscCylinderRow3Middle.Reset();
		_components.qOscCylinderRow3Right.Reset();
    seq.StepCompleteWhen(TRUE);
END_IF        
//***************************************************************************************************   


//***************************************************************************************************     
IF seq.Step(20,TRUE,'<#VYCHODIZA POLOHA - VYPNUTIE DOPRAVNIKOV#>') THEN   
		_components.qEntryFeederRun.Reset();
		_components.qOscConvRun.Reset();
		_components.qOscConvRunReverse.Reset();

	
    seq.StepCompleteWhen(TRUE);
END_IF       
//***************************************************************************************************   


IF (seq.Step(inStepID := seq.RESTORE_STEP_ID,
    inEnabled := TRUE,
    inStepDescription := 'RETURN TO THE START OF THE SEQUENCE')) THEN
    //--------------------------------------------------------	
		refSequenceTask.DoneWhen(TRUE);
    	seq.CompleteSequence();
    //--------------------------------------------------------			
END_IF;



IF refSequenceTask.HandleTaskError() THEN
	
	//here we can decide what to do
	//	refSequenceTask.Restore();

END_IF

seq.Close();
END_METHOD

(*~
	<docu>
		<summary>
		    Custom service (manual, maintenance) logic.
			This method must be implemented in derived class.
		</summary>			
	</docu>	
~*)
METHOD PROTECTED  ServiceMode
IF NOT _config.ControledByVisonSystem THEN
    _components.Designer.Service();
    _components.qEntryFeederRun.Service();
    _components.qOscConvRun.Service();
    _components.qOscConvRunReverse.Service();
    _components.qOscCylinderRow1Left.Service();
    _components.qOscCylinderRow1Middle.Service();
    _components.qOscCylinderRow1Right.Service();
    _components.qOscCylinderRow2Left.Service();
    _components.qOscCylinderRow2Middle.Service();
    _components.qOscCylinderRow2Right.Service();
    _components.qOscCylinderRow3Left.Service();
    _components.qOscCylinderRow3Middle.Service();
    _components.qOscCylinderRow3Right.Service();
	 _components.SideGuard.Service();

END_IF;
END_METHOD

PROPERTY PUBLIC SetSequencesToStep : bool
GET
SetSequencesToStep:=_setSequencesToStep;
END_GET
SET
_setSequencesToStep:=SetSequencesToStep;
END_SET
END_PROPERTY

METHOD PUBLIC SetToDefault : TcoCore.ITcoTaskStatus
SetToDefault := _setToDefaultTask.Invoke();
END_METHOD

PROPERTY SetToDefaultTask : REFERENCE TO TcoFeedingSequenceTask
GET
SetToDefaultTask ref=_setToDefaultTask;
END_GET
END_PROPERTY

PROPERTY PUBLIC SpecificUserData :REFERENCE TO TcoOscilatingConveyorFeeder_PlcToPc
GET
SpecificUserData ref=_specificData.PlcToPcData;
END_GET
END_PROPERTY

(*~
	<docu>
		<summary>
			Gets the status of the MTS Oscilating conveyor feeder. 					
		</summary>			
	</docu>	
~*)
PROPERTY Status : REFERENCE TO TcoOscilatingConveyorFeeder_Status_v_1_x_x
GET
Status REF= _status;
END_GET
END_PROPERTY

METHOD PUBLIC ThrowComponents : TcoCore.ITcoTaskStatus
ThrowComponents := _throwCompoentsTask.Invoke();
END_METHOD

PROPERTY ThrowComponentsTask : REFERENCE TO TcoFeedingSequenceTask
GET
ThrowComponentsTask ref=_throwCompoentsTask;
END_GET
END_PROPERTY

END_FUNCTION_BLOCK

// ---- Abstractions/Components/MtsFeeding/Components/OscilatingConveyorFeeder/TcoOscilatingConveyorFeeder_DesignerSpecificData.TcPOU
FUNCTION_BLOCK TcoOscilatingConveyorFeeder_DesignerSpecificData EXTENDS TcoCognexVision.TcoDesignerRootContainer  
VAR_INPUT
END_VAR
VAR_OUTPUT
END_VAR
VAR
	{attribute wpf [Container(Layout.Stack,"PcToPlc")]}	
	{attribute wpf [Group(Layout.GroupBox)]}
	{attribute addProperty Name "<#PcToPlc#>"}
	PcToPlc:TcoOscilatingConveyorFeeder_PcToPlc ;
	{attribute wpf [Container(Layout.Stack,"PlcToPc")]}	
	{attribute wpf [Group(Layout.GroupBox)]}
	{attribute addProperty Name "<#PlcToPc#>"}
	PlcToPc:TcoOscilatingConveyorFeeder_PlcToPc;
	
END_VAR

PROPERTY PUBLIC PcToPlcData : REFERENCE TO TcoOscilatingConveyorFeeder_PcToPlc
GET
PcToPlcData ref= PcToPlc;
END_GET
END_PROPERTY

PROPERTY PUBLIC PlcToPcData : REFERENCE TO TcoOscilatingConveyorFeeder_PlcToPc
GET
PlcToPcData ref= PlcToPc;
END_GET
END_PROPERTY

END_FUNCTION_BLOCK

// ---- Abstractions/Components/Rework/ReworkInstructionTask.TcPOU
FUNCTION_BLOCK ReworkInstructionTask EXTENDS TcoCore.TcoRemoteTask
VAR
	_data:ReworkData;
END_VAR

SUPER^();

PROPERTY Data : REFERENCE TO ReworkData
GET
Data ref= _data;
END_GET
END_PROPERTY

METHOD Run : REFERENCE TO ReworkInstructionTask
VAR_INPUT
	inEntityId:STRING;
END_VAR
_data.EntityId:=inEntityId;
Run REF= THIS^;
END_METHOD

END_FUNCTION_BLOCK

// ---- Abstractions/Components/TS/EqTransfer/TcoEq2Transfer.TcPOU
{attribute wpf [Container(Layout.Stack)]}
{attribute wpf [Group(Layout.Scroll)]}
FUNCTION_BLOCK TcoEq2Transfer EXTENDS TcoCore.TcoComponent


VAR
	
	_config:TcoEq2Transfer_Config;
	_status:TcoEq2Transfer_Status;
	_control:TcoEq2Transfer_Control;
    _components:TcoEq2TransferComponents:= (Parent := THIS^);
	_handleIncomingPaletteTask:TcoCore.TcoTask(THIS^);
	_handleOutgoingPaletteTask:TcoCore.TcoTask(THIS^);
	_autoTask:TcoCore.TcoTask(THIS^);
	_restoreTask:TcoCore.TcoTask(THIS^);
	
	_progressIncomming:INT;
	_progressOutgoing:INT;

	{attribute 'hide'} 
	_timerIncoming :  TON;
	{attribute 'hide'} 
	_timerOutcoming :  TON;
	
	{attribute 'hide'} 
	_infoTimer :  TON;
    {attribute 'hide'} 
	_errorTimer :  TON;

	_autoProgress: INT;
	
	 {attribute 'hide'} 
	_timerOptional:  TON;
	_mode: eTcoEq2TransferHandlingMode;
END_VAR

_handleIncomingPaletteTask.Enabled := NOT _handleOutgoingPaletteTask.Busy;
IF (_handleIncomingPaletteTask.Execute()) THEN

    IF _config.Configuration = eTcoEq2TransferConfiguration.DoubleInSingleOut THEN
		 IF IsService THEN
		   _mode:=_config.Mode;
	   END_IF
        IncomingPaletteDoubleIn(inMode := _mode,
            refProgress := _progressIncomming,
            refStatus := _status,
            refConfig := _config,
            refTimer := _timerIncoming,
            refTask := _handleIncomingPaletteTask);
    ELSIF _config.Configuration = eTcoEq2TransferConfiguration.SingleInDoubleOut THEN
        IncomingPaletteSingleIn(refProgress := _progressIncomming,
            refStatus := _status,
            refConfig := _config,
            refTimer := _timerIncoming,
            refTask := _handleIncomingPaletteTask);
    END_IF;

    CallTimers(TRUE);
    _handleIncomingPaletteTask.ThrowWhen(_errorTimer.Q);

    Messenger.OnCondition(_infoTimer.Q).Info(_status.ActionDescription);
END_IF;

_handleOutgoingPaletteTask.Enabled := NOT _handleIncomingPaletteTask.Busy;
IF (_handleOutgoingPaletteTask.Execute()) THEN
	IF _config.Configuration = eTcoEq2TransferConfiguration.DoubleInSingleOut THEN
    OutgoingPaletteDoubleIn(refProgress := _progressOutgoing,
        refStatus := _status,
        refConfig := _config,
        refTimer := _timerOutcoming,
        refTask := _handleOutgoingPaletteTask);
   ELSIF _config.Configuration = eTcoEq2TransferConfiguration.SingleInDoubleOut THEN
	   IF IsService THEN
		   _mode:=_config.Mode;
	   END_IF
	   OutgoingPaletteSingleIn(refProgress := _progressOutgoing,
        inMode := _mode,
        refStatus := _status,
        refConfig := _config,
        refTimer := _timerOutcoming,
        refTask := _handleOutgoingPaletteTask);
	END_IF
    CallTimers(TRUE);
    _handleOutgoingPaletteTask.ThrowWhen(_errorTimer.Q);
    Messenger.OnCondition(_infoTimer.Q).Info(_status.ActionDescription);
END_IF;

_autoTask.Enabled := TRUE;
IF (_autoTask.Execute()) THEN

    IF _autoProgress = 0 THEN
        _handleOutgoingPaletteTask.Restore();
    END_IF

    IF _autoProgress = 1 THEN
        IF HandleIncommingPalette().Done THEN
            _autoProgress := _autoProgress + 1;
            _handleOutgoingPaletteTask.Restore();
        END_IF

    END_IF;

    IF _autoProgress = 2 THEN
        IF HandleOutgoingPalette().Done THEN
            _autoProgress := 0;
        end_If;
    END_IF

END_IF;

//*************RESTORE********************

_restoreTask.Enabled := TRUE;

IF _restoreTask.Execute() THEN
    Restore();
	_components.TransferUnit.MoveToHome();
    _restoreTask.DoneWhen(inCondition := _components.TransferUnit.AtHome);
END_IF
//****************************************

METHOD AutomatControl : ITcoTaskStatus
VAR_INPUT
END_VAR
AutomatControl:=_autoTask.Invoke();
END_METHOD

METHOD CallTimers
VAR_INPUT
	inValue : BOOL;
END_VAR
IF   THIS^._config.ErrorTime <> T#0S OR NOT inValue THEN  
_errorTimer(IN := inValue, PT := THIS^._config.ErrorTime);
END_IF;
IF   THIS^._config.InfoTime <>T#0S OR NOT inValue THEN  
_infoTimer(IN := inValue, PT := THIS^._config.InfoTime);
END_IF;
END_METHOD

PROPERTY Components : REFERENCE TO TcoEq2TransferComponents
GET
Components ref=_components;
END_GET
END_PROPERTY


PROPERTY Config : REFERENCE TO TcoEq2Transfer_Config
GET
Config REF= _config;
END_GET
END_PROPERTY

PROPERTY PUBLIC HandleIncomingTask : REFERENCE TO TcoCore.TcoTask
GET
HandleIncomingTask ref= _handleIncomingPaletteTask;
END_GET
END_PROPERTY

METHOD PUBLIC HandleIncommingPalette : TcoCore.ITcoTaskStatus
VAR_INPUT
END_VAR
HandleIncommingPalette:=_handleIncomingPaletteTask.Invoke();
END_METHOD

METHOD PUBLIC HandleOutgoingPalette : TcoCore.ITcoTaskStatus
VAR_INPUT
END_VAR
HandleOutgoingPalette:=_handleOutgoingPaletteTask.Invoke();
END_METHOD

PROPERTY PUBLIC HandleOutgoingTask : REFERENCE TO TcoCore.TcoTask
GET
HandleOutgoingTask ref= _handleOutgoingPaletteTask;
END_GET
END_PROPERTY

METHOD PRIVATE IncomingPaletteDoubleIn
VAR_INPUT
	inMode : eTcoEq2TransferHandlingMode;
	refProgress : REFERENCE TO INT;
	refStatus: REFERENCE TO TcoEq2Transfer_Status;
	refConfig: REFERENCE TO TcoEq2Transfer_Config;
	refTimer: REFERENCE TO TON;
	refTask :  REFERENCE TO TcoCore.TcoTask;
END_VAR

VAR
    _progress    : REFERENCE TO INT;


	_status: REFERENCE TO TcoEq2Transfer_Status;
	_config: REFERENCE TO TcoEq2Transfer_Config;
	_timer: REFERENCE TO TON;
	_task :  REFERENCE TO TcoCore.TcoTask;


END_VAR
_progress REF= refProgress;
_status REF= refStatus;
_config REF= refConfig;
_timer REF= refTimer;
_task REF= refTask;

IF _progress = 0 THEN

    _components.qMotor.Set();
    _components.TransferUnit.Stop();
    //init
    IF   NOT _components.TransferUnit.AtHome AND NOT _components.TransferUnit.AtWork THEN

        IF inMode = eTcoEq2TransferHandlingMode.RecieveDirectWay THEN
            _progress := _progress + 1;
        ELSIF inMode = eTcoEq2TransferHandlingMode.RecieveSideWay THEN
            _progress := 5;
            _timer(IN := FALSE);
        END_IF;
    END_IF;

END_IF;

IF _progress = 1 THEN
    _status.ActionDescription := '<#Handle incoming palette - Wait for pallete at prestopper#>';

    IF _components.iStopperMainTransfer.IsTrue THEN
        _progress := 5;
        _timer(IN := FALSE);
    ELSIF _components.iPreStopperMainTransfer.IsTrue THEN
        _progress := _progress + 1;
        _timer(IN := FALSE);
    END_IF
END_IF;

IF _progress = 2 THEN
    _status.ActionDescription := '<#Handle incoming palette - Check transfer unit status#>';

    _timer(IN := _components.iStopperMainTransfer.IsFalse AND
            _components.iMainTransferIsEmpty.IsTrue AND
            NOT _components.TransferUnit.AtHome AND
            NOT _components.TransferUnit.AtWork,
        PT := _config.StabilisationTime);

    IF _components.iStopperMainTransfer.IsFalse AND
        _components.iMainTransferIsEmpty.IsTrue AND
        NOT _components.TransferUnit.AtHome AND
        NOT _components.TransferUnit.AtWork AND
        _timer.Q THEN
        _timer(IN := FALSE);
        _progress := _progress + 1;
    END_IF
END_IF;

IF _progress = 3 THEN
    _status.ActionDescription := '<#Handle incoming palette - Open prestoper#>';
    IF _components.iPreStopperMainTransfer.IsTrue THEN
        _components.qPreStopperMainTransfer.Set();
    END_IF;

    _timer(IN := NOT _components.iPreStopperMainTransfer.Signal, PT := _config.StabilisationTime);

    IF _components.qPreStopperMainTransfer.IsTrue AND _timer.Q THEN
        _components.qPreStopperMainTransfer.Reset();
        _timer(IN := FALSE);
        _progress := _progress + 1;

    END_IF;
END_IF;

IF _progress = 4 THEN
    _status.ActionDescription := '<#Handle incoming palette - Waiting for pallet at stopper - Main Transfer#>';
    _timer(IN := _components.iStopperMainTransfer.IsTrue, PT := _config.StabilisationTime);
    IF _components.iStopperMainTransfer.IsTrue AND _timer.Q THEN
        _progress := 10;
        _timer(IN := FALSE);
    END_IF;
END_IF;

IF _progress = 5 THEN
    _status.ActionDescription := '<#Handle incoming palette - Waiting for pallet at side transfer#>';

    IF _components.iStopperSideTransfer.IsTrue THEN
        _progress := 8;
        _timer(IN := FALSE);
    ELSIF _components.iPrestopperSideTransfer.IsTrue THEN
        _progress := _progress + 1;
        _timer(IN := FALSE);
    END_IF
END_IF;

IF _progress = 6 THEN

    _timer(IN := _components.iStopperSideTransfer.IsFalse AND
            _components.iSideTransferIsEmpty.IsTrue AND
            NOT _components.TransferUnit.AtHome AND
            NOT _components.TransferUnit.AtWork,
        PT := _config.StabilisationTime);

    _status.ActionDescription := '<#Handle incoming palette - Check transfer unit status#>';

    IF _components.iStopperSideTransfer.IsFalse AND
        _components.iSideTransferIsEmpty.IsTrue AND
        NOT _components.TransferUnit.AtHome AND
        NOT _components.TransferUnit.AtWork AND
        _timer.Q THEN
        _timer(IN := FALSE);
        _progress := _progress + 1;
    END_IF
END_IF;

IF _progress = 7 THEN
    _status.ActionDescription := '<#Handle incoming palette - Open side prestoper#>';
    IF _components.iPreStopperSideTransfer.IsTrue THEN
        _components.qPreStopperSideTransfer.Set();
    END_IF;

    _timer(IN := NOT _components.iPreStopperSideTransfer.Signal, PT := _config.StabilisationTime);

    IF _components.iPreStopperSideTransfer.IsFalse AND _timer.Q THEN
        _components.qPreStopperSideTransfer.Reset();
        _timer(IN := FALSE);
        _progress := _progress + 1;

    END_IF;
END_IF;

IF _progress = 8 THEN
    _status.ActionDescription := '<#Handle incoming palette - Waiting for pallet at stopper - Side Transfer#>';
    _timer(IN := _components.iStopperSideTransfer.Signal, PT := _config.StabilisationTime);
    IF _components.iStopperSideTransfer.IsTrue AND _timer.Q THEN
        _progress := _progress + 1;
    END_IF;

END_IF;

IF _progress = 9 THEN
    _status.ActionDescription := '<#Handle incoming palette - Wait Main transfer is empty#>';
    _timer(IN := _components.iMainTransferIsEmpty.Signal, PT := _config.StabilisationTime);
    IF ((_components.iMainTransferIsEmpty.IsTrue AND _timer.Q) AND_THEN _components.TransferUnit.MoveToWork().Done) THEN
        _progress := _progress + 1;
    END_IF;
END_IF;

IF _progress = 10 THEN
    _status.ActionDescription := '<#Handle incoming palette - Wait for pallete in Main transfer#>';
    _timer(IN := (*_components.iSideTransferIsEmpty.Signal AND*) NOT _components.iMainTransferIsEmpty.Signal, PT := _config.StabilisationTime);
    IF ((*_components.iSideTransferIsEmpty.IsTrue AND*) _components.iMainTransferIsEmpty.IsFalse AND _timer.Q) THEN
        _progress := _progress + 1;
    END_IF;
END_IF;

IF _progress = 11 THEN
    _status.ActionDescription := '<#Handle incoming palette - Wait for pallete in main transfer#>';
    IF _components.iStopperMainTransfer.IsTrue AND _components.iMainTransferIsEmpty.IsFalse THEN
        _status.ActionDescription := '<#Done#>';
        _task.DoneWhen(TRUE);
        _progress := 0;
    END_IF;
END_IF;
END_METHOD

METHOD PRIVATE IncomingPaletteSingleIn
VAR_INPUT
	refProgress : REFERENCE TO INT;
	refStatus: REFERENCE TO TcoEq2Transfer_Status;
	refConfig: REFERENCE TO TcoEq2Transfer_Config;
	refTimer: REFERENCE TO TON;
	refTask :  REFERENCE TO TcoCore.TcoTask;
END_VAR

VAR
    _progress    : REFERENCE TO INT;


	_status: REFERENCE TO TcoEq2Transfer_Status;
	_config: REFERENCE TO TcoEq2Transfer_Config;
	_timer: REFERENCE TO TON;
	_task :  REFERENCE TO TcoCore.TcoTask;


END_VAR
_progress REF= refProgress;
_status REF= refStatus;
_config REF= refConfig;
_timer REF= refTimer;
_task REF= refTask;

IF _progress = 0 THEN

    _components.qMotor.Set();

    _components.TransferUnit.Stop();

    IF NOT _components.TransferUnit.AtHome AND NOT _components.TransferUnit.AtWork THEN
        _progress := _progress + 1;
        _timer(IN := FALSE);
        _timerOptional(IN := FALSE);
    END_IF;

END_IF;

IF _progress = 1 THEN

    IF _config.Configuration = eTcoEq2TransferConfiguration.SingleInDoubleOutNoPrestopper THEN
        _progress := 5;
    ELSIF _config.Configuration = eTcoEq2TransferConfiguration.SingleInDoubleOut THEN
        _progress := _progress + 1;
    END_IF;

    _timer(IN := FALSE);
END_IF;

IF _progress = 2 THEN
    _status.ActionDescription := '<#Handle incoming palette - Waiting for pallet at stopper#>';
    _timer(IN := _components.iStopperMainTransfer.IsTrue, PT := _config.StabilisationTime);

    IF _components.iStopperMainTransfer.IsTrue AND _timer.q THEN
        _progress := 5;
        _timer(IN := FALSE);
        _timerOptional(IN := FALSE);

    ELSIF _components.iPreStopperMainTransfer.IsTrue THEN
        _progress := _progress + 1;
        _timer(IN := FALSE);
    END_IF
END_IF;

IF _progress = 3 THEN

    _timer(IN := _components.iStopperMainTransfer.IsFalse AND
            _components.iMainTransferIsEmpty.IsTrue AND
            NOT _components.TransferUnit.AtHome AND
            NOT _components.TransferUnit.AtWork,
        PT := _config.StabilisationTime);

    Messenger.Info('<#Handle incoming palette - Check transfer unit status#>');

    IF _components.iStopperMainTransfer.IsFalse AND
        _components.iMainTransferIsEmpty.IsTrue AND
        NOT _components.TransferUnit.AtHome AND
        NOT _components.TransferUnit.AtWork AND
        _timer.Q THEN
        _timer(IN := FALSE);
        _progress := _progress + 1;
    END_IF
END_IF;

IF _progress = 4 THEN
    _status.ActionDescription := '<#Handle incoming palette - Open prestoper#>';
    IF _components.iPreStopperMainTransfer.IsTrue THEN
        _components.qPreStopperMainTransfer.Set();
    END_IF;

    _timer(IN := NOT _components.iPreStopperMainTransfer.Signal, PT := _config.StabilisationTime);

    IF _components.qPreStopperMainTransfer.IsTrue AND _timer.Q THEN
        _components.qPreStopperMainTransfer.Reset();
        _timer(IN := FALSE);
        _timerOptional(IN := FALSE);
        _progress := _progress + 1;

    END_IF;
END_IF;

IF _progress = 5 THEN
    _status.ActionDescription := '<#Handle incoming palette - Waiting for pallet at stopper - Entry Transfer#>';
    _timer(IN := _components.iStopperMainTransfer.IsTrue, PT := _config.StabilisationTime);
    _timerOptional(IN := TRUE, PT := _config.StabilisationTime * 5);

    IF _components.iStopperMainTransfer.IsTrue AND _timer.Q THEN
        _progress := _progress + 1;
        _timer(IN := FALSE);
    ELSIF _components.iStopperMainTransfer.IsFalse AND _timer.Q THEN
        _progress := 0;
    END_IF

END_IF;

IF _progress = 6 THEN
    _status.ActionDescription := '<#Handle incoming palette - Wait for pallete in workposition#>';
    IF _components.iStopperMainTransfer.IsTrue AND _components.iMainTransferIsEmpty.IsFalse THEN
        _status.ActionDescription := '<#Done#>';

        _task.DoneWhen(TRUE);
        _progress := 0;
    END_IF;
END_IF;
END_METHOD

PROPERTY PUBLIC Mode : reference to eTcoEq2TransferHandlingMode
GET
Mode ref= _mode;
END_GET
END_PROPERTY

METHOD PRIVATE OutgoingPaletteDoubleIn
VAR_INPUT
	refProgress : REFERENCE TO INT;
	refStatus: REFERENCE TO TcoEq2Transfer_Status;
	refConfig: REFERENCE TO TcoEq2Transfer_Config;
	refTimer: REFERENCE TO TON;
	refTask :  REFERENCE TO TcoCore.TcoTask;
END_VAR

VAR
    _progress    : REFERENCE TO INT;


	_status: REFERENCE TO TcoEq2Transfer_Status;
	_config: REFERENCE TO TcoEq2Transfer_Config;
	_timer: REFERENCE TO TON;
	_task :  REFERENCE TO TcoCore.TcoTask;

	_timerOptional: TON;

END_VAR
_progress REF= refProgress;
_status REF= refStatus;
_config REF= refConfig;
_timer REF= refTimer;
_task REF= refTask;
IF _progress = 0 THEN
    //init
	_components.qMotor.Set();
    _progress := _progress + 1;
END_IF;

IF _progress = 1 THEN
    _status.ActionDescription := '<#Handle outgoing palette - Transfer unit home#>';

    IF _components.iWipaMainTransfer.IsFalse AND_THEN _components.TransferUnit.MoveToHome().Done THEN
        _progress := _progress + 1;
        _timer(IN := FALSE);
    END_IF

END_IF;

IF _progress = 2 THEN
    _status.ActionDescription := '<#Handle outgoing palette - Wait to transfer unit is empty#>';

    _timer(IN := NOT _components.iStopperMainTransfer.Signal AND _components.iMainTransferIsEmpty.Signal, PT := _config.StabilisationTime);

    IF (_components.iStopperMainTransfer.IsFalse AND _components.iMainTransferIsEmpty.IsTrue AND _timer.Q) THEN
        _progress := _progress + 1;
        _timer(IN := FALSE);
    END_IF;
END_IF;

IF _progress = 3 THEN
    _status.ActionDescription := '<#Handle outgoing palette - Transfer unit to middle position#>';
    _components.TransferUnit.Stop();
    _timer(IN := TRUE, PT := _config.StabilisationTime);

    IF (NOT _components.TransferUnit.AtHome AND NOT _components.TransferUnit.AtWork) THEN
        _progress := 10;
        _timer(IN := FALSE);
    END_IF;
END_IF;

IF _progress = 10 THEN
	_components.qMotor.Reset();
    _status.ActionDescription := '<#Handle outgoing palette - Done#>';
    _task.DoneWhen(TRUE);
    _progress := 0;

END_IF;
END_METHOD

METHOD PRIVATE OutgoingPaletteSingleIn
VAR_INPUT
    inMode : eTcoEq2TransferHandlingMode;
    refProgress : REFERENCE TO INT;
    refStatus : REFERENCE TO TcoEq2Transfer_Status;
    refConfig : REFERENCE TO TcoEq2Transfer_Config;
    refTimer : REFERENCE TO TON;
    refTask : REFERENCE TO TcoCore.TcoTask;
END_VAR

VAR
    _progress : REFERENCE TO INT;

    _status : REFERENCE TO TcoEq2Transfer_Status;
    _config : REFERENCE TO TcoEq2Transfer_Config;
    _timer : REFERENCE TO TON;
    _task : REFERENCE TO TcoCore.TcoTask;

    _timerOptional : TON;

END_VAR
_progress REF= refProgress;
_status REF= refStatus;
_config REF= refConfig;
_timer REF= refTimer;
_task REF= refTask;

IF _progress = 0 THEN
    _status.ActionDescription := '<#Handle outgoing palette - Init#>';

    _components.qMotor.Set();
    _progress := _progress + 1;
END_IF;

IF _progress = 1 THEN
	 _status.ActionDescription := '<#Handle outgoing palette - Send Direct/Send Side#>';
    IF inMode = eTcoEq2TransferHandlingMode.SendDirectWay THEN
        IF _components.iWipaMainTransfer.IsFalse AND_THEN _components.TransferUnit.MoveToHome().Done THEN
            _progress := _progress + 1;
            _timer(IN := FALSE);
        END_IF
    ELSIF inMode = eTcoEq2TransferHandlingMode.SendSideWay THEN

        _progress := 4;
        _timer(IN := FALSE);

    END_IF;
END_IF;

IF _progress = 2 THEN
	 _status.ActionDescription := '<#Handle outgoing palette - Check Main transfer is empty#>';

    _timer(IN := NOT _components.iStopperMainTransfer.Signal AND _components.iMainTransferIsEmpty.Signal,
        PT := _config.StabilisationTime);

    IF (_components.iStopperMainTransfer.IsFalse AND _components.iMainTransferIsEmpty.IsTrue AND _timer.Q) THEN
        _progress := _progress + 1;
        _timer(IN := FALSE);
    END_IF;
END_IF;

IF _progress = 3 THEN
    _status.ActionDescription := '<#Handle outgoing palette - Wait Trasnfer unit at Middle position (not home,not work)#>';
    _components.TransferUnit.Stop();
    _timer(IN := TRUE, PT := _config.StabilisationTime);

    IF NOT _components.TransferUnit.AtHome AND NOT _components.TransferUnit.AtWork THEN
        _progress := 10;
        _timer(IN := FALSE);
    END_IF;
END_IF;

IF _progress = 4 THEN
    _status.ActionDescription := '<#Handle outgoing palette - Wait Side transfer is empty#>';
    _timer(IN := _components.iSideTransferIsEmpty.Signal, PT := _config.StabilisationTime);
    IF ((_components.iSideTransferIsEmpty.IsTrue AND _timer.Q) AND_THEN _components.TransferUnit.MoveToWork().Done) THEN
        _progress := _progress + 1;
    END_IF;
END_IF;

IF _progress = 5 THEN
    _status.ActionDescription := '<#Handle outgoing palette - Wait for pallete in side transfer#>';
    _timer(IN := _components.iMainTransferIsEmpty.Signal AND NOT _components.iSideTransferIsEmpty.Signal, PT := _config.StabilisationTime);
    IF (_components.iMainTransferIsEmpty.IsTrue AND _components.iSideTransferIsEmpty.IsFalse AND _timer.Q) THEN
        _progress := _progress + 1;
    END_IF;
END_IF;

IF _progress = 6 THEN
    _status.ActionDescription := '<#Handle outgoing palette - Transfer unit middle position#>';
    IF _components.iWipaSideTransfer.IsFalse THEN
        _components.TransferUnit.Stop();
        IF NOT _components.TransferUnit.AtHome AND NOT _components.TransferUnit.AtWork THEN
            _progress := 10;
        END_IF;
    END_IF;
END_IF;

IF _progress = 10 THEN
    _components.qMotor.Reset();
    _status.ActionDescription := '<#Handle outgoing palette - Done#>';
    _task.DoneWhen(TRUE);
    _progress := 0;

END_IF;
END_METHOD

(*~
	<docu>
		<summary>
			Restores this instance to the Ready state. Can be called explicitly or from within one of the restore mechanisms.	
		</summary>			
	</docu>	
~*)
METHOD  Restore : ITcoRestorable
_handleIncomingPaletteTask.Restore();
_handleOutgoingPaletteTask.Restore();
_autoTask.Restore();
CallTimers(FALSE);
_timerOptional(IN:=FALSE);

_components.qMotor.Reset();
_progressIncomming:=0;
_progressOutgoing:=0;

IF _config.Configuration = eTcoEq2TransferConfiguration.DoubleInSingleOut THEN
	Components.qPreStopperMainTransfer.Reset();
	Components.qPrestopperSideTransfer.Reset();
ELSIF _config.Configuration = eTcoEq2TransferConfiguration.SingleInDoubleOut THEN
	Components.qPreStopperMainTransfer.Reset();
END_IF;
THIS^.Messenger.UnPin();
END_METHOD

PROPERTY PUBLIC RestoreTask : REFERENCE TO TcoCore.TcoTask
GET
RestoreTask ref= _restoreTask;
END_GET
END_PROPERTY

(*~
	<docu>
		<summary>
		    Custom service (manual, maintenance) logic.
			This method must be implemented in derived class.
		</summary>			
	</docu>	
~*)
METHOD PROTECTED  ServiceMode
_components.qPreStopperMainTransfer.Service();
_components.qPrestopperSideTransfer.Service();
_components.qMotor.Service();

_components.TransferUnit.Service();
END_METHOD


PROPERTY Status : REFERENCE TO TcoEq2Transfer_Status
GET
Status REF= _status;
END_GET
END_PROPERTY

PROPERTY TransferIsEmpty : bool
GET
TransferIsEmpty:=Components.iMainTransferIsEmpty.Signal AND Components.iSideTransferIsEmpty.Signal AND not Components.TransferUnit.AtHome and not Components.TransferUnit.AtWork;
END_GET
END_PROPERTY

END_FUNCTION_BLOCK

// ---- Abstractions/Components/TS/RotaryTrabsferWithLift/TcoLiftingRotaryTransfer.TcPOU
{attribute wpf [Container(Layout.Stack)]}
{attribute wpf [Group(Layout.Scroll)]}
FUNCTION_BLOCK TcoLiftingRotaryTransfer EXTENDS TcoCore.TcoComponent


VAR
	
	_config:TcoLiftingRotaryTransfer_Config;
	_status:TcoLiftingRotaryTransfer_Status;
	_control:TcoLiftingRotaryTransfer_Control;
    _components:TcoLiftingRotaryTransferComponents:= (Parent := THIS^);
	_handleIncomingPaletteTask:TcoCore.TcoTask(THIS^);
	_handleOutgoingPaletteTask:TcoCore.TcoTask(THIS^);
	_autoTask:TcoCore.TcoTask(THIS^);
	_restoreTask:TcoCore.TcoTask(THIS^);
	
	_progressIncomming:INT;
	_progressOutgoing:INT;

	{attribute 'hide'} 
	_timerIncoming :  TON;
	{attribute 'hide'} 
	_timerOutcoming :  TON;
	
	{attribute 'hide'} 
	_infoTimer :  TON;
    {attribute 'hide'} 
	_errorTimer :  TON;

	_autoProgress: INT;
	
	_timerOptional: TON;

END_VAR

_handleIncomingPaletteTask.Enabled := NOT _handleOutgoingPaletteTask.Busy;
IF (_handleIncomingPaletteTask.Execute()) THEN
    IncomingPalette(refProgress := _progressIncomming,
        refStatus := _status,
        refConfig := _config,
        refTimer := _timerIncoming,
        refTask := _handleIncomingPaletteTask);

    CallTimers(TRUE);
    _handleIncomingPaletteTask.ThrowWhen(_errorTimer.Q);

    Messenger.OnCondition(_infoTimer.Q).Info(_status.ActionDescription);
END_IF;

_handleOutgoingPaletteTask.Enabled := NOT _handleIncomingPaletteTask.Busy;
IF (_handleOutgoingPaletteTask.Execute()) THEN
    OutgoingPalette(refProgress := _progressOutgoing,
        refStatus := _status,
        refConfig := _config,
        refTimer := _timerOutcoming,
        refTask := _handleOutgoingPaletteTask);

    CallTimers(TRUE);
    _handleOutgoingPaletteTask.ThrowWhen(_errorTimer.Q);
    Messenger.OnCondition(_infoTimer.Q).Info(_status.ActionDescription);
END_IF;

_autoTask.Enabled := TRUE;
IF (_autoTask.Execute()) THEN

    IF _autoProgress = 0 THEN
        _handleOutgoingPaletteTask.Restore();
		_autoProgress:=_autoProgress+1;
    END_IF

    IF _autoProgress = 1 THEN
        IF HandleIncommingPalette().Done THEN
            _autoProgress := _autoProgress + 1;
            _handleOutgoingPaletteTask.Restore();
        END_IF

    END_IF;

    IF _autoProgress = 2 THEN
        IF HandleOutgoingPalette().Done THEN
            _autoProgress := 0;
        end_If;
    END_IF

END_IF;

//*************RESTORE********************

_restoreTask.Enabled := TRUE;

IF _restoreTask.Execute() THEN
    Restore();

    IF _config.InvertLifting THEN
      IF _components.Lift.MoveToWork().Done AND_THEN _components.RotaryUnit.MoveToWork().Done THEN
            _restoreTask.DoneWhen(inCondition := TRUE);

        END_IF
    ELSE
         IF components.Lift.MoveToHome().Done AND_THEN components.RotaryUnit.MoveToHome().Done  THEN
            _restoreTask.DoneWhen(inCondition := TRUE);

        END_IF
    END_IF
END_IF
//****************************************

METHOD AutomatControl : ITcoTaskStatus
VAR_INPUT
END_VAR
AutomatControl:=_autoTask.Invoke();
END_METHOD

METHOD CallTimers
VAR_INPUT
	inValue : BOOL;
END_VAR
IF   THIS^._config.ErrorTime <> T#0S OR NOT inValue THEN  
_errorTimer(IN := inValue, PT := THIS^._config.ErrorTime);
END_IF;
IF   THIS^._config.InfoTime <>T#0S OR NOT inValue THEN  
_infoTimer(IN := inValue, PT := THIS^._config.InfoTime);
END_IF;
END_METHOD

PROPERTY Components : REFERENCE TO TcoLiftingRotaryTransferComponents
GET
Components ref=_components;
END_GET
END_PROPERTY


PROPERTY Config : REFERENCE TO TcoLiftingRotaryTransfer_Config
GET
Config REF= _config;
END_GET
END_PROPERTY

PROPERTY PUBLIC HandleIncomingTask : REFERENCE TO TcoCore.TcoTask
GET
HandleIncomingTask ref= _handleIncomingPaletteTask;
END_GET
END_PROPERTY

METHOD PUBLIC HandleIncommingPalette : TcoCore.ITcoTaskStatus
VAR_INPUT
END_VAR
HandleIncommingPalette:=_handleIncomingPaletteTask.Invoke();
END_METHOD

METHOD PUBLIC HandleOutgoingPalette : TcoCore.ITcoTaskStatus
VAR_INPUT
END_VAR
HandleOutgoingPalette:=_handleOutgoingPaletteTask.Invoke();
END_METHOD

PROPERTY PUBLIC HandleOutgoingTask : REFERENCE TO TcoCore.TcoTask
GET
HandleOutgoingTask ref= _handleOutgoingPaletteTask;
END_GET
END_PROPERTY

METHOD PRIVATE IncomingPalette
VAR_INPUT
	refProgress : REFERENCE TO INT;
	refStatus: REFERENCE TO TcoLiftingRotaryTransfer_Status;
	refConfig: REFERENCE TO TcoLiftingRotaryTransfer_Config;
	refTimer: REFERENCE TO TON;
	refTask :  REFERENCE TO TcoCore.TcoTask;
END_VAR

VAR
    _progress    : REFERENCE TO INT;


	_status: REFERENCE TO TcoLiftingRotaryTransfer_Status;
	_config: REFERENCE TO TcoLiftingRotaryTransfer_Config;
	_timer: REFERENCE TO TON;
	_task :  REFERENCE TO TcoCore.TcoTask;
	
	
END_VAR
_progress REF= refProgress;
_status REF= refStatus;
_config REF= refConfig;
_timer REF= refTimer;
_task REF= refTask;

IF _progress = 0 THEN
	_components.qMotor.Set();
    _progress := _progress + 1;

END_IF

IF _progress = 1 THEN
    _status.ActionDescription := '<#Handle incoming palette - Wait for pallete at prestopper#>';
	
    CallTimers(FALSE);
    IF _components.iStopper.IsTrue THEN
        _progress := 4;

    ELSIF _components.iPrestopper.IsTrue THEN
        _progress := _progress + 1;
        _timer(IN := FALSE);
		_timerOptional(IN:=FALSE);
    END_IF;
END_IF

IF _progress = 2 THEN
    _status.ActionDescription := '<#Handle incoming palette - Check status of workposition #>';
    _timer(IN := NOT _Components.iStopper.Signal AND NOT Components.qPrestopper.Signal, PT := _config.StabilisationTime);
    _timerOptional(in := TRUE, Pt := T#2S);

    IF _config.InvertLifting AND
        Components.iStopper.IsFalse AND
        Components.iTransferIsEmpty.IsTrue AND
        Components.qStopper.IsFalse AND
        Components.Lift.AtWork AND 
		Components.RotaryUnit.AtWork AND
        _timer.Q THEN
        _timer(IN := FALSE);
		_timerOptional(IN:=FALSE);
      	_progress := _progress+1;
    ELSIF NOT _config.InvertLifting AND
        Components.iStopper.IsFalse AND
        Components.iTransferIsEmpty.IsTrue AND
        Components.qStopper.IsFalse AND
        Components.Lift.AtHome AND
		Components.RotaryUnit.AtHome AND
        _timer.Q THEN
        _timer(IN := FALSE);
		_timerOptional(IN:=FALSE);
      	_progress := _progress+1;

    ELSIF Components.iStopper.IsTrue AND _timerOptional.Q AND Components.iTransferIsEmpty.IsFalse AND Components.qStopper.IsTrue THEN
         _timer(IN := FALSE);
		_timerOptional(IN:=FALSE);
      	_progress := _progress+1;

    END_IF

END_IF

IF _progress = 3 THEN
    _status.ActionDescription := '<#Handle incoming palette - Open prestopper#>';

    IF _components.iPrestopper.IsTrue THEN
        _components.qPrestopper.Set();
    END_IF;

    _timer(IN := NOT _components.iPrestopper.Signal, PT := _config.StabilisationTime);

    IF _components.qPrestopper.IsTrue AND _timer.Q THEN
        _components.qPrestopper.Reset();
        _timer(IN := FALSE);
        _progress := _progress + 1;
    END_IF
END_IF

IF _progress = 4 THEN
    _status.ActionDescription := '<#Handle incoming palette - Wait for pallete in workposition#>';

    IF _components.iStopper.IsTrue THEN
        _task.DoneWhen(TRUE);
		_progress:=0;
    END_IF;
END_IF;
END_METHOD

METHOD PRIVATE OutgoingPalette
VAR_INPUT
	refProgress : REFERENCE TO INT;
	refStatus: REFERENCE TO TcoLiftingRotaryTransfer_Status;
	refConfig: REFERENCE TO TcoLiftingRotaryTransfer_Config;
	refTimer: REFERENCE TO TON;
	refTask :  REFERENCE TO TcoCore.TcoTask;
END_VAR

VAR
    _progress    : REFERENCE TO INT;


	_status: REFERENCE TO TcoLiftingRotaryTransfer_Status;
	_config: REFERENCE TO TcoLiftingRotaryTransfer_Config;
	_timer: REFERENCE TO TON;
	_task :  REFERENCE TO TcoCore.TcoTask;


END_VAR
_progress REF= refProgress;
_status REF= refStatus;
_config REF= refConfig;
_timer REF= refTimer;
_task REF= refTask;

IF _progress = 0 THEN
	_components.qMotor.Set();

    _progress := _progress + 1;

END_IF

IF _progress = 1 THEN
    _status.ActionDescription := '<#Handle outgoing palette - Check lift rotary unit position)#>';
    IF _config.InvertLifting THEN
        _timer(IN := _Components.RotaryUnit.AtHome, PT := _config.StabilisationTime);

        IF _components.RotaryUnit.MoveToHome().Done AND_THEN _timer.q AND_THEN _components.Lift.MoveToHome().Done THEN
            _progress := _progress + 1;
            _timer(IN := FALSE);
        END_IF
    ELSE
        _timer(IN := Components.RotaryUnit.AtWork, PT := _config.StabilisationTime);
        IF _components.RotaryUnit.MoveToWork().Done AND_THEN _timer.q AND_THEN _components.Lift.MoveToWork().Done THEN
            _progress := _progress + 1;
            _timer(IN := FALSE);
        END_IF;
    END_IF
END_IF

IF _progress = 2 THEN
    _status.ActionDescription := '<#Handle outgoing palette - Open stopper to send palette#>';

    IF _components.iWipa.IsFalse THEN
        _components.qStopper.Set();
    END_IF

    _timer(IN := _components.qStopper.Signal AND NOT _components.iStopper.Signal, PT := _config.StabilisationTime);
    _timerOptional(IN := TRUE, Pt := T#2S);

    IF (_components.qStopper.IsTrue AND _timer.Q) OR (_components.qStopper.IsFalse AND _components.iStopper.IsFalse AND _timerOptional.q) THEN
        _components.qStopper.Reset();
        _progress := _progress + 1;
        _timer(IN := FALSE);
    END_IF;
END_IF;

IF _progress = 3 THEN
    Messenger.Info('Handle outgoing palette - Wait for transfer is empty');
    _timer(IN := _components.iTransferIsEmpty.Signal AND NOT _components.iStopper.Signal, PT := _config.StabilisationTime);
    IF (_components.iTransferIsEmpty.IsTrue AND _components.iStopper.IsFalse AND _timer.Q) THEN
        _progress := _progress + 1;
        _timer(IN := FALSE);
    END_IF;
END_IF;

IF _progress = 4 THEN
	 Messenger.Info('Handle outgoing palette - Cylinders to wait positions ');
	 _components.qMotor.Reset();
  IF _config.InvertLifting THEN
        IF _components.Lift.MoveToWork().Done AND_THEN _components.RotaryUnit.MoveToWork().Done THEN
            _task.DoneWhen(TRUE);
        _progress := 0;
        END_IF;
    ELSE
        IF _components.Lift.MoveToHome().Done AND_THEN _components.RotaryUnit.MoveToHome().Done THEN
            _task.DoneWhen(TRUE);
        _progress := 0;
        END_IF;
    END_IF;

END_IF;
END_METHOD

(*~
	<docu>
		<summary>
			Restores this instance to the Ready state. Can be called explicitly or from within one of the restore mechanisms.	
		</summary>			
	</docu>	
~*)
METHOD  Restore : ITcoRestorable
_handleIncomingPaletteTask.Restore();
_handleOutgoingPaletteTask.Restore();
_autoTask.Restore();
CallTimers(FALSE);

_components.qStopper.Reset();
_components.qPrestopper.Reset();
_components.qMotor.Reset();
_progressIncomming:=0;
_progressOutgoing:=0;
THIS^.Messenger.UnPin();
END_METHOD

PROPERTY PUBLIC RestoreTask : REFERENCE TO TcoCore.TcoTask
GET
RestoreTask ref= _restoreTask;
END_GET
END_PROPERTY

(*~
	<docu>
		<summary>
		    Custom service (manual, maintenance) logic.
			This method must be implemented in derived class.
		</summary>			
	</docu>	
~*)
METHOD PROTECTED  ServiceMode
_components.RotaryUnit.Service();
_components.Lift.Service();
_components.qPrestopper.Service();
_components.qStopper.Service();
_components.qMotor.Service();
END_METHOD


PROPERTY Status : REFERENCE TO TcoLiftingRotaryTransfer_Status
GET
Status REF= _status;
END_GET
END_PROPERTY

END_FUNCTION_BLOCK

// ---- Abstractions/Components/TS/RotaryTransfer/TcoRotaryTransfer.TcPOU
{attribute wpf [Container(Layout.Stack)]}
{attribute wpf [Group(Layout.Scroll)]}
FUNCTION_BLOCK TcoRotaryTransfer EXTENDS TcoCore.TcoComponent


VAR
	
	_config:TcoRotaryTransfer_Config;
	_status:TcoRotaryTransfer_Status;
	_control:TcoRotaryTransfer_Control;
    _components:TcoRotaryTransferComponents:= (Parent := THIS^);
	_handleIncomingPaletteTask:TcoCore.TcoTask(THIS^);
	_handleOutgoingPaletteTask:TcoCore.TcoTask(THIS^);
	_autoTask:TcoCore.TcoTask(THIS^);
	_restoreTask:TcoCore.TcoTask(THIS^);
	
	_progressIncomming:INT;
	_progressOutgoing:INT;

	{attribute 'hide'} 
	_timerIncoming :  TON;
	{attribute 'hide'} 
	_timerOutcoming :  TON;
	
	{attribute 'hide'} 
	_infoTimer :  TON;
    {attribute 'hide'} 
	_errorTimer :  TON;

	_autoProgress: INT;
END_VAR

_handleIncomingPaletteTask.Enabled := NOT _handleOutgoingPaletteTask.Busy;
IF (_handleIncomingPaletteTask.Execute()) THEN
    IncomingPalette(refProgress := _progressIncomming,
        refStatus := _status,
        refConfig := _config,
        refTimer := _timerIncoming,
        refTask := _handleIncomingPaletteTask);
		
	CallTimers(TRUE);
	_handleIncomingPaletteTask.ThrowWhen(_errorTimer.Q);

	Messenger.OnCondition(_infoTimer.Q).Info(_status.ActionDescription); 
END_IF;


_handleOutgoingPaletteTask.Enabled := NOT _handleIncomingPaletteTask.Busy;
IF (_handleOutgoingPaletteTask.Execute()) THEN
    OutgoingPalette(refProgress := _progressOutgoing,
        refStatus := _status,
        refConfig := _config,
        refTimer := _timerOutcoming,
        refTask := _handleOutgoingPaletteTask);
		
	CallTimers(TRUE);
	_handleOutgoingPaletteTask.ThrowWhen(_errorTimer.Q);
	Messenger.OnCondition(_infoTimer.Q).Info(_status.ActionDescription); 
END_IF;


_autoTask.Enabled := TRUE;
IF (_autoTask.Execute()) THEN
	
	IF _autoProgress =0 THEN
		_handleOutgoingPaletteTask.Restore();
	END_IF
	
	IF _autoProgress = 1  THEN
		IF  HandleIncommingPalette().Done THEN
			_autoProgress:=_autoProgress+1;
			_handleOutgoingPaletteTask.Restore();
		END_IF
		
	END_IF;
	IF _autoProgress = 2  THEN
		IF HandleOutgoingPalette().Done THEN
			_autoProgress:=0;
		end_If;
	END_IF
 
END_IF;

//*************RESTORE********************

_restoreTask.Enabled := TRUE;
IF _restoreTask.Execute() THEN
	Restore();
	_restoreTask.DoneWhen(inCondition:=_components.RotaryUnit.AtHome);
END_IF
//****************************************

METHOD AutomatControl : ITcoTaskStatus
VAR_INPUT
END_VAR
AutomatControl:=_autoTask.Invoke();
END_METHOD

METHOD CallTimers
VAR_INPUT
	inValue : BOOL;
END_VAR
IF   THIS^._config.ErrorTime <> T#0S OR NOT inValue THEN  
_errorTimer(IN := inValue, PT := THIS^._config.ErrorTime);
END_IF;
IF   THIS^._config.InfoTime <>T#0S OR NOT inValue THEN  
_infoTimer(IN := inValue, PT := THIS^._config.InfoTime);
END_IF;
END_METHOD

PROPERTY Components : REFERENCE TO TcoRotaryTransferComponents
GET
Components ref=_components;
END_GET
END_PROPERTY


PROPERTY Config : REFERENCE TO TcoRotaryTransfer_Config
GET
Config REF= _config;
END_GET
END_PROPERTY

PROPERTY PUBLIC HandleIncomingTask : REFERENCE TO TcoCore.TcoTask
GET
HandleIncomingTask ref= _handleIncomingPaletteTask;
END_GET
END_PROPERTY

METHOD PUBLIC HandleIncommingPalette : TcoCore.ITcoTaskStatus
VAR_INPUT
END_VAR
HandleIncommingPalette:=_handleIncomingPaletteTask.Invoke();
END_METHOD

METHOD PUBLIC HandleOutgoingPalette : TcoCore.ITcoTaskStatus
VAR_INPUT
END_VAR
HandleOutgoingPalette:=_handleOutgoingPaletteTask.Invoke();
END_METHOD

PROPERTY PUBLIC HandleOutgoingTask : REFERENCE TO TcoCore.TcoTask
GET
HandleOutgoingTask ref= _handleOutgoingPaletteTask;
END_GET
END_PROPERTY

METHOD PRIVATE IncomingPalette
VAR_INPUT
	refProgress : REFERENCE TO INT;
	refStatus: REFERENCE TO TcoRotaryTransfer_Status;
	refConfig: REFERENCE TO TcoRotaryTransfer_Config;
	refTimer: REFERENCE TO TON;
	refTask :  REFERENCE TO TcoCore.TcoTask;
END_VAR

VAR
    _progress    : REFERENCE TO INT;


	_status: REFERENCE TO TcoRotaryTransfer_Status;
	_config: REFERENCE TO TcoRotaryTransfer_Config;
	_timer: REFERENCE TO TON;
	_task :  REFERENCE TO TcoCore.TcoTask;


END_VAR
_progress REF= refProgress;
_status REF= refStatus;
_config REF= refConfig;
_timer REF= refTimer;
_task REF= refTask;

IF _progress = 0 THEN
	_components.qMotor.Set();
    _progress := _progress + 1;

END_IF

IF _progress = 1 THEN
    _status.ActionDescription := '<#Handle outgoing palette - Wait for pallete at prestopper#>';

    CallTimers(FALSE);
    IF _components.iStopper.IsTrue THEN
        _progress := 3;

    ELSIF _components.iPrestopper.IsTrue THEN
        _progress := _progress + 1;
        _timer(IN := FALSE);
    END_IF;
END_IF

IF _progress = 2 THEN
    _status.ActionDescription := '<#Handle incoming palette - Check status of workposition #>';
    _timer(IN := NOT _components.iStopper.Signal AND NOT _components.qPrestopper.Signal, PT := _config.StabilisationTime);

    IF _components.iStopper.IsFalse AND _components.qStopper.IsFalse AND (_components.RotaryUnit.AtHome) AND _timerIncoming.Q THEN
        _timer(IN := FALSE);
        _progress := _progress + 1;
    END_IF
END_IF

IF _progress = 3 THEN
    _status.ActionDescription := '<#Handle incoming palette - Open prestopper#>';

    IF _components.iPrestopper.IsTrue THEN
        _components.qPrestopper.Set();
    END_IF;

    _timer(IN := NOT _components.iPrestopper.Signal, PT := _config.StabilisationTime);

    IF _components.qPrestopper.IsTrue AND _timer.Q THEN
        _components.qPrestopper.Reset();
        _timer(IN := FALSE);
        _progress := _progress + 1;
    END_IF
END_IF

IF _progress = 4 THEN
    _status.ActionDescription := '<#Handle incoming palette - Wait for pallete in workposition#>';

    IF _components.iStopper.IsTrue THEN
        _task.DoneWhen(TRUE);
		_progress:=0;
    END_IF;
END_IF;
END_METHOD

METHOD PRIVATE OutgoingPalette
VAR_INPUT
	refProgress : REFERENCE TO INT;
	refStatus: REFERENCE TO TcoRotaryTransfer_Status;
	refConfig: REFERENCE TO TcoRotaryTransfer_Config;
	refTimer: REFERENCE TO TON;
	refTask :  REFERENCE TO TcoCore.TcoTask;
END_VAR

VAR
    _progress    : REFERENCE TO INT;


	_status: REFERENCE TO TcoRotaryTransfer_Status;
	_config: REFERENCE TO TcoRotaryTransfer_Config;
	_timer: REFERENCE TO TON;
	_task :  REFERENCE TO TcoCore.TcoTask;

	_timerOptional: TON;

END_VAR
_progress REF= refProgress;
_status REF= refStatus;
_config REF= refConfig;
_timer REF= refTimer;
_task REF= refTask;

IF _progress = 0 THEN
	 _status.ActionDescription := '<#Handle outgoing palette - Init#>';
	_components.qMotor.Set();
    _progress := _progress + 1;

END_IF

IF _progress = 1 THEN
    _status.ActionDescription := '<#Handle outgoing palette - rotary unit to work #>';

    IF _components.RotaryUnit.MoveToWork().Done THEN
        _progress := _progress + 1;
        _timer(IN := FALSE);
    END_IF;
END_IF

IF _progress = 2 THEN
    _status.ActionDescription := '<#Handle outgoing palette - Open stopper to send palette#>';

    IF _components.iWipa.IsFalse THEN
        _components.qStopper.Set();
    END_IF

    _timer(IN := _components.qStopper.Signal AND NOT _components.iStopper.Signal, PT := _config.StabilisationTime);
    _timerOptional(IN := TRUE, Pt := T#2S);

    IF (_components.qStopper.IsTrue AND _timer.Q) OR (_components.qStopper.IsFalse AND _components.iStopper.IsFalse AND _timerOptional.q) THEN
        _components.qStopper.Reset();
        _progress := _progress + 1;
        _timer(IN := FALSE);
    END_IF;
END_IF;

IF _progress = 3 THEN
    Messenger.Info('Handle outgoing palette - Wait for transfer is empty (send to next)');
    _timer(IN := _components.iTransferIsEmpty.Signal AND NOT _components.iStopper.Signal, PT := _config.StabilisationTime);
    IF (Components.iTransferIsEmpty.IsTrue AND Components.iStopper.IsFalse AND _timer.Q) THEN
        _progress := _progress + 1;
        _timer(IN := FALSE);
    END_IF;
END_IF;

IF _progress = 4 THEN
   Messenger.Info('Handle outgoing palette - rotary unit to home');
    IF (Components.RotaryUnit.MoveToHome().Done) THEN
		_components.qMotor.Reset();
          _task.DoneWhen(TRUE);
		  _progress:=0;
    END_IF;
END_IF;
END_METHOD

(*~
	<docu>
		<summary>
			Restores this instance to the Ready state. Can be called explicitly or from within one of the restore mechanisms.	
		</summary>			
	</docu>	
~*)
METHOD  Restore : ITcoRestorable
_handleIncomingPaletteTask.Restore();
_handleOutgoingPaletteTask.Restore();
_autoTask.Restore();
CallTimers(FALSE);
_components.RotaryUnit.MoveHomeTask.Invoke();
_components.qStopper.Reset();
_components.qPrestopper.Reset();
_components.qMotor.Reset();
_progressIncomming:=0;
_progressOutgoing:=0;
THIS^.Messenger.UnPin();
END_METHOD

PROPERTY PUBLIC RestoreTask : REFERENCE TO TcoCore.TcoTask
GET
RestoreTask ref= _restoreTask;
END_GET
END_PROPERTY

(*~
	<docu>
		<summary>
		    Custom service (manual, maintenance) logic.
			This method must be implemented in derived class.
		</summary>			
	</docu>	
~*)
METHOD PROTECTED  ServiceMode
_components.RotaryUnit.Service();
_components.qPrestopper.Service();
_components.qStopper.Service();
END_METHOD


PROPERTY Status : REFERENCE TO TcoRotaryTransfer_Status
GET
Status REF= _status;
END_GET
END_PROPERTY

END_FUNCTION_BLOCK

// ---- Abstractions/Components/TS/WorkPosition/TcoTransferSystemComponent.TcPOU
{attribute wpf [Container(Layout.Stack)]}
{attribute wpf [Group(Layout.Scroll)]}
FUNCTION_BLOCK TcoTransferSystemComponent EXTENDS TcoCore.TcoComponent

VAR
    _config : TcoTransferSystem_Config;
    _status : TcoTransferSystem_Status;
    _control : TcoTransferSystem_Control;
    _components : TcoTransferSystemComponents := (Parent := THIS^);
    _handleIncomingPaletteTask : TcoCore.TcoTask(THIS^);
    _handleOutgoingPaletteTask : TcoCore.TcoTask(THIS^);
    _restoreTask : TcoCore.TcoTask(THIS^);

    _progressIncomming : INT;
    _progressOutgoing : INT;

    {attribute 'hide'}
    _timerIncoming : TON;
    {attribute 'hide'}
    _timerOutcoming : TON;

    {attribute 'hide'}
    _infoTimer : TON;
    {attribute 'hide'}
    _errorTimer : TON;

    _timerOptional : TON;

END_VAR

_handleIncomingPaletteTask.Enabled := TRUE;
IF (_handleIncomingPaletteTask.Execute()) THEN
    IncomingPalette(refProgress := _progressIncomming,
        refStatus := _status,
        refConfig := _config,
        refTimer := _timerIncoming,
        refTask := _handleIncomingPaletteTask);

    CallTimers(TRUE);
    _handleIncomingPaletteTask.ThrowWhen(_errorTimer.Q);
    Messenger.OnCondition(_infoTimer.Q).Info(_status.ActionDescription);
END_IF;

_handleOutgoingPaletteTask.Enabled := TRUE;
IF (_handleOutgoingPaletteTask.Execute()) THEN
    OutgoingPalette(refProgress := _progressOutgoing,
        refStatus := _status,
        refConfig := _config,
        refTimer := _timerOutcoming,
        refTask := _handleOutgoingPaletteTask);

    CallTimers(TRUE);
    _handleOutgoingPaletteTask.ThrowWhen(_errorTimer.Q);
    Messenger.OnCondition(_infoTimer.Q).Info(_status.ActionDescription);
END_IF;

//*************RESTORE********************

_restoreTask.Enabled := TRUE;

IF _restoreTask.Execute() THEN
    Restore();
    IF _config.HasPositionUnit THEN
        _restoreTask.DoneWhen(inCondition := _components.PositionUnit.AtHome);
	 ELSE
        _restoreTask.DoneWhen(inCondition :=TRUE);
    END_IF;
END_IF
//****************************************

METHOD CallTimers
VAR_INPUT
	inValue : BOOL;
END_VAR
IF   THIS^._config.ErrorTime <> T#0S OR NOT inValue THEN  
_errorTimer(IN := inValue, PT := THIS^._config.ErrorTime);
END_IF;
IF   THIS^._config.InfoTime <>T#0S OR NOT inValue THEN  
_infoTimer(IN := inValue, PT := THIS^._config.InfoTime);
END_IF;
END_METHOD

PROPERTY Components : REFERENCE TO TcoTransferSystemComponents
GET
Components ref=_components;
END_GET
END_PROPERTY


PROPERTY Config : REFERENCE TO TcoTransferSystem_Config
GET
Config REF= _config;
END_GET
END_PROPERTY

PROPERTY PUBLIC HandleIncomingTask : REFERENCE TO TcoCore.TcoTask
GET
HandleIncomingTask ref= _handleIncomingPaletteTask;
END_GET
END_PROPERTY

METHOD PUBLIC HandleIncommingPalette : TcoCore.ITcoTaskStatus
VAR_INPUT
END_VAR
HandleIncommingPalette:=_handleIncomingPaletteTask.Invoke();
END_METHOD

METHOD PUBLIC HandleOutgoingPalette : TcoCore.ITcoTaskStatus
VAR_INPUT
END_VAR
HandleOutgoingPalette:=_handleOutgoingPaletteTask.Invoke();
END_METHOD

PROPERTY PUBLIC HandleOutgoingTask : REFERENCE TO TcoCore.TcoTask
GET
HandleOutgoingTask ref= _handleOutgoingPaletteTask;
END_GET
END_PROPERTY

METHOD PRIVATE IncomingPalette
VAR_INPUT
	refProgress : REFERENCE TO INT;
	refStatus: REFERENCE TO TcoTransferSystem_Status;
	refConfig: REFERENCE TO TcoTransferSystem_Config;
	refTimer: REFERENCE TO TON;
	refTask :  REFERENCE TO TcoCore.TcoTask;
END_VAR

VAR
    _progress    : REFERENCE TO INT;


	_status: REFERENCE TO TcoTransferSystem_Status;
	_config: REFERENCE TO TcoTransferSystem_Config;
	_timer: REFERENCE TO TON;
	_task :  REFERENCE TO TcoCore.TcoTask;


END_VAR
_progress REF= refProgress;
_status REF= refStatus;
_config REF= refConfig;
_timer REF= refTimer;
_task REF=refTask;

	
IF _progress = 0 THEN
	_status.ActionDescription := '<#Handle incoming palette - Handle incoming palette start (Check position unit position)#>'; 
	IF _Components.PositionUnit.AtHome OR  NOT _config.HasPositionUnit THEN
		_progress := _progress + 1;	
	END_IF;
END_IF

IF _progress = 1 THEN
	_status.ActionDescription := '<#Handle incoming palette - Wait for pallete at prestopper#>';

	CallTimers(FALSE);
	IF _components.iStopper.IsTrue THEN
		_progress:=4;
	
	ELSIF _components.iPrestopper.IsTrue THEN
		_progress := _progress + 1;
		_timer(IN:=FALSE);
	END_IF;
END_IF

IF _progress = 2 THEN
	_status.ActionDescription := '<#Handle incoming palette - Check status of workposition #>';
	_timer(IN:=NOT _components.iStopper.Signal AND  NOT _components.qPrestopper.Signal ,PT:=_config.StabilisationTime);
	
	IF _components.iStopper.IsFalse
		AND _components.qStopper.IsFalse
		AND (_components.PositionUnit.AtHome or not _config.HasPositionUnit) 
		AND _timerIncoming.Q THEN
		_timer(IN:=FALSE);
		_progress := _progress + 1;
	END_IF
END_IF

IF _progress = 3 THEN
	_status.ActionDescription := '<#Handle incoming palette - Open prestopper#>';
	
	IF _components.iPrestopper.IsTrue THEN
		_components.qPrestopper.Set();
	END_IF;
	
	_timer(IN:=NOT _components.iPrestopper.Signal ,PT:=_config.StabilisationTime );
	
	IF _components.qPrestopper.IsTrue
		AND _timer.Q THEN
		_components.qPrestopper.Reset();
		_timer(IN:=FALSE);
		_progress := _progress + 1;
	END_IF
END_IF

	
IF _progress = 4 THEN
    _status.ActionDescription:='<#Handle incoming palette - Wait for pallete in workposition#>';	

	IF _components.iStopper.IsTrue AND NOT  _config.HasPositionUnit	 THEN
	 	_task.DoneWhen(TRUE);
	ELSIF _components.iStopper.IsTrue  THEN
	 	 	_task.DoneWhen(TRUE);
	END_IF;
END_IF;
END_METHOD

METHOD PRIVATE OutgoingPalette
VAR_INPUT
	refProgress : REFERENCE TO INT;
	refStatus: REFERENCE TO TcoTransferSystem_Status;
	refConfig: REFERENCE TO TcoTransferSystem_Config;
	refTimer: REFERENCE TO TON;
	refTask :  REFERENCE TO TcoCore.TcoTask;
END_VAR

VAR
    _progress    : REFERENCE TO INT;


	_status: REFERENCE TO TcoTransferSystem_Status;
	_config: REFERENCE TO TcoTransferSystem_Config;
	_timer: REFERENCE TO TON;
	_task :  REFERENCE TO TcoCore.TcoTask;



END_VAR
_progress REF= refProgress;
_status REF= refStatus;
_config REF= refConfig;
_timer REF= refTimer;
_task REF=refTask;

IF _progress = 0 THEN

	_progress := _progress + 1;	

END_IF
	
IF _progress = 1 THEN
	_status.ActionDescription := '<#Handle outgoing palette - Start (Check position unit position)#>';
 	IF _config.HasPositionUnit THEN
		_components.PositionUnit.MoveToHome();
	END_IF
	IF _components.PositionUnit.AtHome AND  _config.HasPositionUnit THEN
		_progress := _progress + 1;	
		_timer(IN:=FALSE);
	ELSIF NOT _config.HasPositionUnit THEN
		_progress := _progress + 1;	
		_timer(IN:=FALSE);
	END_IF;
END_IF



IF _progress = 2 THEN
    _status.ActionDescription:='<#Handle outgoing palette - Open stopper to send palette to next station#>';	
	
	 IF _components.iWipa.IsFalse THEN
        _components.qStopper.Set();
    END_IF

    _timer(IN := _components.qStopper.Signal AND NOT _components.iStopper.Signal, PT := _config.StabilisationTime);
	_timerOptional(IN:=TRUE,Pt:=T#2S);
	
    IF (_components.qStopper.IsTrue AND _timer.Q)
		OR (_components.qStopper.IsFalse AND _components.iStopper.IsFalse AND _timerOptional.q) THEN
     	 _components.qStopper.Reset();
    	_task.DoneWhen(TRUE);
	END_IF;
END_IF;
END_METHOD

(*~
	<docu>
		<summary>
			Restores this instance to the Ready state. Can be called explicitly or from within one of the restore mechanisms.	
		</summary>			
	</docu>	
~*)
METHOD  Restore : ITcoRestorable
_handleIncomingPaletteTask.Restore();
_handleOutgoingPaletteTask.Restore();
CallTimers(FALSE);
_components.PositionUnit.MoveHomeTask.Invoke();
_components.qStopper.Reset();
_components.qPrestopper.Reset();
_progressIncomming:=0;
_progressOutgoing:=0;
THIS^.Messenger.UnPin();
END_METHOD

PROPERTY PUBLIC RestoreTask : REFERENCE TO TcoCore.TcoTask
GET
RestoreTask ref= _restoreTask;
END_GET
END_PROPERTY

(*~
	<docu>
		<summary>
		    Custom service (manual, maintenance) logic.
			This method must be implemented in derived class.
		</summary>			
	</docu>	
~*)
METHOD PROTECTED  ServiceMode
_components.PositionUnit.Service();
_components.qPrestopper.Service();
_components.qStopper.Service();
END_METHOD


PROPERTY Status : REFERENCE TO TcoTransferSystem_Status
GET
Status REF= _status;
END_GET
END_PROPERTY

END_FUNCTION_BLOCK

// ---- Abstractions/Components/WrappedComponent/WrappedComponentExample.TcPOU
FUNCTION_BLOCK WrappedComponentExample EXTENDS TcoCore.TcoComponent


VAR_OUTPUT
END_VAR
VAR
	_config:WrappedComponentExample_Config;
	_status:WrappedComponentExample_Status;
	_control:WrappedComponentExample_Control;
    _components:WrappedComponentsExample:= (Parent := THIS^);
	_throwTask:TcoCore.TcoTask(THIS^);
	_restoreTask:TcoCore.TcoTask(THIS^);

END_VAR

_throwTask();
_restoreTask.Enabled:=true;
_restoreTask();

PROPERTY Components : REFERENCE TO WrappedComponentsExample
GET
Components ref=_components;
END_GET
END_PROPERTY

(*~
	<docu>
		<summary>
			Restores this instance to the Ready state. Can be called explicitly or from within one of the restore mechanisms.	
		</summary>			
	</docu>	
~*)
METHOD  Restore : ITcoRestorable
END_METHOD

(*~
	<docu>
		<summary>
		    Custom service (manual, maintenance) logic.
			This method must be implemented in derived class.
		</summary>			
	</docu>	
~*)
METHOD PROTECTED  ServiceMode
END_METHOD

END_FUNCTION_BLOCK

// ---- Abstractions/CUBase/CUBase.TcPOU
{attribute addProperty ShortName ""}
FUNCTION_BLOCK ABSTRACT CUBase EXTENDS TcoCore.TcoObject IMPLEMENTS ICUBase

VAR
    _cuId        : eStations;
    _processData : ProcessDataManager(THIS^);
	_groupInspection : TcoInspectors.TcoInspectionGroup(THIS^);
	{attribute addProperty Name "<#STATUS INFO#>"}
    _statusInfo  : CUBaseStatusInfo := (Parent := THIS^);
	_operatorInfo : OperatorInfo := (Parent := THIS^);
	_settings  : CUBaseSettings := (Parent := THIS^);
	_toggle: TcoUtilities.TcoBlinker(THIS^);
	_recurringFails:CuBaseRecurringFailures:=(Parent:=THIS^);
	_productionPlaner:ProductionPlaner(THIS^);
	_internalData : REFERENCE TO InternalStorage;	
	
	{attribute clr [ReadOnly()]}
	{attribute clr [RenderIgnore()]}
	_readyForOperations : BOOL;
END_VAR

(*~
	<docu>
		<summary>
			Controls `automatic` mode of `CU00x`.
		</summary>
	</docu>
~*)
METHOD  Automat
VAR_INPUT
END_VAR
(*
	Enable condition to start `automatTask`.
	Modify according your needs.
	[! 
	THIS IS NOT SAFETY CONDITION. THE SAFETY OF PRESONNEL AND EQUIPMENT MUST BE ENSURED BY ADDITIONAL MEANS 
	TO COMPLY WITH REGULATIONS
	]
*)


AutomatTask.Task.Enabled :=  AutomatTask.Task.Busy  XOR
							(GroundTask.GroundDone AND NOT AutomatTask.Task.Busy AND THIS^.Technology.AllowAutomat(inCuId:=CuId));

(*
	Invokes `groundTask` from technology object.
*)

IF(Technology.AutomatAllTask.Execute()) THEN AutomatTask.Task.Invoke(); END_IF;

IF(Technology.ForceStepMode()) THEN
 	AutomatTask.ModeController.Mode := eSequencerMode.StepMode;
END_IF
END_METHOD

PROPERTY ABSTRACT AutomatTask : REFERENCE TO CUBaseAutomat
GET
END_GET
END_PROPERTY

PROPERTY  CreateEntityTask : TcoCore.ITcoTaskStatus
GET
CreateEntityTask := _processData._createTask;
END_GET
END_PROPERTY

PROPERTY CuId : eStations
GET
CuId := _cuId;
END_GET
SET
_cuId := CuId;
END_SET
END_PROPERTY

PROPERTY  DeleteEntityTask : TcoCore.ITcoTaskStatus
GET
DeleteEntityTask := _processData._deleteTask;
END_GET
END_PROPERTY

METHOD DoesBelong : BOOL
DoesBelong := THIS^.ProcessDataManager.Data.EntityHeader.NextStation = THIS^.CuId;
END_METHOD

METHOD EntityFlowCloseForOperations : TcoCore.ITcoTaskStatus
VAR_IN_OUT
	Header : CuHeader; 
END_VAR
THIS^.FlagCloseEntity(Header);
EntityFlowCloseForOperations := THIS^.ProcessDataManager.Update(ProcessDataManager.Data._EntityId);
END_METHOD

METHOD EntityFlowCreateNew : TcoCore.ITcoTaskStatus
VAR_INPUT
	EntityId : STRING(255);	
END_VAR
VAR_IN_OUT
	Header : CuHeader;
END_VAR
THIS^.FlagCreateNewEntity(EntityId, Header);
EntityFlowCreateNew := THIS^.ProcessDataManager.Create(EntityId);
END_METHOD

METHOD EntityFlowDiscard : TcoCore.ITcoTaskStatus
VAR_INPUT
	EntityId : STRING(255);	
END_VAR
VAR_IN_OUT	
	Header : CuHeader; 
END_VAR
THIS^.FlagThrowAwayEntity(Header);
EntityFlowDiscard := THIS^.ProcessDataManager.Update(EntityId);
END_METHOD

METHOD EntityFlowFinalize : TcoCore.ITcoTaskStatus
VAR_IN_OUT
	Header : CuHeader; 
END_VAR
THIS^.FlagFinishEntity(Header);
EntityFlowFinalize := THIS^.ProcessDataManager.Update(ProcessDataManager.Data._EntityId);
END_METHOD

METHOD EntityFlowOpenForOperations : TcoCore.ITcoTaskStatus
VAR_INPUT
	Identifier : STRING(255);	
END_VAR
VAR_IN_OUT
	Header : CuHeader;
END_VAR
EntityFlowOpenForOperations := THIS^.ProcessDataManager.Read(Identifier);
THIS^.FlagOpenEntity(Identifier, Header);
END_METHOD

PROPERTY  ExistEntityTask : TcoCore.ITcoTaskStatus
GET
ExistEntityTask := _processData._idExistsTask;
END_GET
END_PROPERTY

METHOD PRIVATE FlagCloseEntity : BOOL
VAR_IN_OUT
	Header : CuHeader; 
END_VAR
THIS^.ProcessDataManager.Data.EntityHeader.LastStation := THIS^.CuId;

IF(THIS^.ProcessDataManager.Data.EntityHeader.Results.Result = TcoInspectors.eOverallResult.Failed) THEN	
	THIS^.ProcessDataManager.Data.EntityHeader.NextStation := Header.NextOnFailed;
ELSIF(THIS^.ProcessDataManager.Data.EntityHeader.Results.Result = TcoInspectors.eOverallResult.Passed) THEN
	THIS^.ProcessDataManager.Data.EntityHeader.NextStation := Header.NextOnPassed;
ELSIF(THIS^.ProcessDataManager.Data.EntityHeader.Results.Result = TcoInspectors.eOverallResult.InProgress) THEN
	THIS^.ProcessDataManager.Data.EntityHeader.NextStation := Header.NextOnPassed;
END_IF

THIS^.ProcessDataManager.Data.EntityHeader.OpenOn := eStations.NONE;
Header.CycleTime := THIS^._statusInfo.CurrentCycleTime;
Header.CleanLoopTime := THIS^._statusInfo.CurrentCleanCycleTime;
Header.OperationsEnded := Context.RealTimeClock.NowLocal();
Header.Operator := _operatorInfo.UserName;
END_METHOD

METHOD PRIVATE FlagCreateNewEntity : BOOL
VAR_INPUT
	Identifier : STRING(255);	
END_VAR
VAR_IN_OUT
	Header : CuHeader;
END_VAR
THIS^.ProcessDataManager.Data.EntityHeader.Results.Result := TcoInspectors.eOverallResult.InProgress;
THIS^.ProcessDataManager.Data._EntityId := Identifier;
THIS^.ProcessDataManager.Data.EntityHeader.WasReset := FALSE;
END_METHOD

METHOD PRIVATE FlagFinishEntity : BOOL
VAR_IN_OUT
	Header : CuHeader; 
END_VAR
THIS^.ProcessDataManager.Data.EntityHeader.LastStation := THIS^.CuId;

IF(THIS^.ProcessDataManager.Data.EntityHeader.Results.Result = TcoInspectors.eOverallResult.InProgress) THEN
	THIS^.ProcessDataManager.Data.EntityHeader.Results.Result := TcoInspectors.eOverallResult.Passed;
END_IF

IF(THIS^.ProcessDataManager.Data.EntityHeader.Results.Result = TcoInspectors.eOverallResult.Failed) THEN	
	THIS^.ProcessDataManager.Data.EntityHeader.NextStation := Header.NextOnFailed;
ELSIF(THIS^.ProcessDataManager.Data.EntityHeader.Results.Result = TcoInspectors.eOverallResult.Passed) THEN
	THIS^.ProcessDataManager.Data.EntityHeader.NextStation := Header.NextOnPassed;
END_IF

THIS^.ProcessDataManager.Data.EntityHeader.OpenOn := eStations.NONE;

Header.CycleTime := THIS^._statusInfo.CurrentCycleTime;
Header.CleanLoopTime := THIS^._statusInfo.CurrentCleanCycleTime;
Header.OperationsEnded := Context.RealTimeClock.NowLocal();
Header.Operator := _operatorInfo.UserName;
END_METHOD

